KUKA KRL program: f1_Kuka_APT219T03S19.SRC

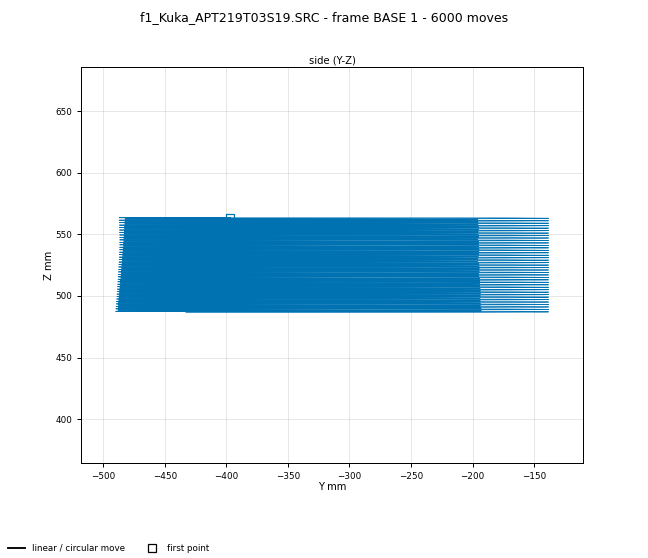
[picture p0: tool path of f1_Kuka_APT219T03S19.SRC in frame BASE 1, 6000 of 6001 moves have a stored position in this frame; points joined in program order, loops and branches not executed]
&ACCESS RVP
&REL 2
&PARAM TEMPLATE = C:\KRC\Roboter\Template\vorgabe
&PARAM EDITMASK = *
DEF f1_Kuka_APT219T03S19()


;FOLD INI;%{PE}%V3.2.0,%MKUKATPBASIS,%CINIT,%VCOMMON,%P
  ;FOLD BAS INI;%{E}%V3.2.0,%MKUKATPBASIS,%CINIT,%VINIT,%P
    GLOBAL INTERRUPT DECL 3 WHEN $STOPMESS==TRUE DO IR_STOPM ( )
    INTERRUPT ON 3
    BAS (#INITMOV,0 )
  ;ENDFOLD (BAS INI)
  ;FOLD USER INI;%{E}%V3.2.0,%MKUKATPUSER,%CINIT,%VINIT,%P
    ;Make your modifications here
  ;ENDFOLD (USER INI)
;ENDFOLD (INI)


;*** Make Null PTP Move
  PTP $pos_act

;*** Auto Load The Correct TOOL Data
  $tool=tool_data[3]

;*** Auto Load The Correct BASE Data
  $base=base_data[1]

  $ADVANCE = 5

;*** Restate Last Velocity
MMPM(30000.0)
SetRPM(6000)
LIN {X 0.052,Y -396.888,Z 563.591,A 0.000,B 0.000,C 90.000,E1 286.315} C_DIS
LIN {X 0.069,Y -413.808,Z 563.580,A 0.000,B 0.000,C 90.000,E1 284.356} C_DIS
LIN {X -0.094,Y -425.703,Z 563.572,A 0.000,B 0.000,C 90.000,E1 283.008} C_DIS
LIN {X 0.164,Y -434.823,Z 563.566,A 0.000,B 0.000,C 90.000,E1 281.895} C_DIS
LIN {X 0.106,Y -443.464,Z 563.560,A 0.000,B 0.000,C 90.000,E1 280.838} C_DIS
LIN {X -0.094,Y -449.609,Z 563.556,A 0.000,B 0.000,C 90.000,E1 280.074} C_DIS
LIN {X -0.070,Y -457.217,Z 563.550,A 0.000,B 0.000,C 90.000,E1 279.029} C_DIS
LIN {X -0.024,Y -464.281,Z 563.544,A 0.000,B 0.000,C 90.000,E1 277.992} C_DIS
LIN {X 0.173,Y -470.590,Z 563.539,A 0.000,B 0.000,C 90.000,E1 276.947} C_DIS
LIN {X -0.087,Y -476.108,Z 563.533,A 0.000,B 0.000,C 90.000,E1 275.967} C_DIS
LIN {X -0.149,Y -479.640,Z 563.529,A 0.000,B 0.000,C 90.000,E1 275.220} C_DIS
LIN {X 0.002,Y -481.624,Z 563.526,A 0.000,B 0.000,C 90.000,E1 274.702} C_DIS
LIN {X 0.124,Y -483.330,Z 563.523,A 0.000,B 0.000,C 90.000,E1 274.188} C_DIS
LIN {X -0.189,Y -484.732,Z 563.521,A 0.000,B 0.000,C 90.000,E1 273.726} C_DIS
LIN {X -0.041,Y -485.835,Z 563.518,A 0.000,B 0.000,C 90.000,E1 273.212} C_DIS
LIN {X 0.144,Y -486.619,Z 563.515,A 0.000,B 0.000,C 90.000,E1 272.694} C_DIS
LIN {X -0.175,Y -486.999,Z 563.512,A 0.000,B 0.000,C 90.000,E1 272.236} C_DIS
LIN {X 0.015,Y -486.990,Z 563.510,A 0.000,B 0.000,C 90.000,E1 271.718} C_DIS
LIN {X 0.189,Y -486.484,Z 563.507,A 0.000,B 0.000,C 90.000,E1 271.203} C_DIS
LIN {X -0.120,Y -485.459,Z 563.504,A 0.000,B 0.000,C 90.000,E1 270.745} C_DIS
LIN {X 0.053,Y -483.968,Z 563.501,A 0.000,B 0.000,C 90.000,E1 270.229} C_DIS
LIN {X 0.221,Y -481.805,Z 563.499,A 0.000,B 0.000,C 90.000,E1 269.714} C_DIS
LIN {X -0.102,Y -478.951,Z 563.496,A 0.000,B 0.000,C 90.000,E1 269.255} C_DIS
LIN {X 0.035,Y -475.279,Z 563.493,A 0.000,B 0.000,C 90.000,E1 268.740} C_DIS
LIN {X 0.149,Y -470.579,Z 563.490,A 0.000,B 0.000,C 90.000,E1 268.224} C_DIS
LIN {X -0.010,Y -467.817,Z 563.489,A 0.000,B 0.000,C 90.000,E1 267.993} C_DIS
LIN {X -0.053,Y -461.679,Z 563.486,A 0.000,B 0.000,C 90.000,E1 267.535} C_DIS
LIN {X 0.032,Y -454.984,Z 563.484,A 0.000,B 0.000,C 90.000,E1 267.135} C_DIS
LIN {X -0.209,Y -447.920,Z 563.482,A 0.000,B 0.000,C 90.000,E1 266.846} C_DIS
LIN {X 0.025,Y -440.647,Z 563.481,A 0.000,B 0.000,C 90.000,E1 266.560} C_DIS
LIN {X 0.215,Y -432.943,Z 563.480,A 0.000,B 0.000,C 90.000,E1 266.331} C_DIS
LIN {X -0.106,Y -424.380,Z 563.479,A 0.000,B 0.000,C 90.000,E1 266.216} C_DIS
LIN {X -0.080,Y -413.364,Z 563.478,A 0.000,B 0.000,C 90.000,E1 266.102} C_DIS
LIN {X 0.171,Y -408.029,Z 563.478,A 0.000,B 0.000,C 90.000,E1 266.045} C_DIS
LIN {X 0.041,Y -180.922,Z 563.478,A 0.000,B 0.000,C 90.000,E1 266.045} C_DIS
LIN {X 0.082,Y -180.869,Z 563.472,A 0.000,B 0.000,C 90.000,E1 265.008} C_DIS
LIN {X -0.015,Y -178.930,Z 563.443,A 0.000,B 0.000,C 90.000,E1 259.803} C_DIS
LIN {X 0.023,Y -175.977,Z 563.415,A 0.000,B 0.000,C 90.000,E1 254.700} C_DIS
LIN {X -0.032,Y -175.468,Z 563.410,A 0.000,B 0.000,C 90.000,E1 253.866} C_DIS
LIN {X 0.025,Y -172.217,Z 563.387,A 0.000,B 0.000,C 90.000,E1 249.571} C_DIS
LIN {X 0.002,Y -171.693,Z 563.382,A 0.000,B 0.000,C 90.000,E1 248.720} C_DIS
LIN {X 0.078,Y -167.287,Z 563.353,A 0.000,B 0.000,C 90.000,E1 243.512} C_DIS
LIN {X 0.011,Y -166.663,Z 563.348,A 0.000,B 0.000,C 90.000,E1 242.666} C_DIS
LIN {X -0.073,Y -162.646,Z 563.324,A 0.000,B 0.000,C 90.000,E1 238.329} C_DIS
LIN {X -0.011,Y -161.335,Z 563.314,A 0.000,B 0.000,C 90.000,E1 236.548} C_DIS
LIN {X 0.033,Y -157.330,Z 563.290,A 0.000,B 0.000,C 90.000,E1 232.110} C_DIS
LIN {X -0.034,Y -155.312,Z 563.275,A 0.000,B 0.000,C 90.000,E1 229.461} C_DIS
LIN {X 0.003,Y -151.668,Z 563.250,A 0.000,B 0.000,C 90.000,E1 224.960} C_DIS
LIN {X 0.047,Y -150.534,Z 563.240,A 0.000,B 0.000,C 90.000,E1 223.137} C_DIS
LIN {X -0.022,Y -147.259,Z 563.215,A 0.000,B 0.000,C 90.000,E1 218.624} C_DIS
LIN {X 0.034,Y -145.285,Z 563.194,A 0.000,B 0.000,C 90.000,E1 214.945} C_DIS
LIN {X 0.068,Y -142.386,Z 563.164,A 0.000,B 0.000,C 90.000,E1 209.411} C_DIS
LIN {X -0.010,Y -141.364,Z 563.148,A 0.000,B 0.000,C 90.000,E1 206.668} C_DIS
LIN {X -0.032,Y -139.344,Z 563.112,A 0.000,B 0.000,C 90.000,E1 200.174} C_DIS
LIN {X -0.026,Y -139.013,Z 563.102,A 0.000,B 0.000,C 90.000,E1 198.308} C_DIS
LIN {X -0.031,Y -138.342,Z 563.055,A 0.000,B 0.000,C 90.000,E1 189.905} C_DIS
LIN {X -0.011,Y -139.397,Z 563.008,A 0.000,B 0.000,C 90.000,E1 181.489} C_DIS
LIN {X 0.043,Y -141.299,Z 562.972,A 0.000,B 0.000,C 90.000,E1 174.951} C_DIS
LIN {X 0.000,Y -142.661,Z 562.957,A 0.000,B 0.000,C 90.000,E1 172.186} C_DIS
LIN {X -0.050,Y -145.005,Z 562.931,A 0.000,B 0.000,C 90.000,E1 167.589} C_DIS
LIN {X -0.061,Y -147.631,Z 562.911,A 0.000,B 0.000,C 90.000,E1 163.921} C_DIS
LIN {X 0.017,Y -150.261,Z 562.890,A 0.000,B 0.000,C 90.000,E1 160.242} C_DIS
LIN {X 0.031,Y -153.661,Z 562.870,A 0.000,B 0.000,C 90.000,E1 156.613} C_DIS
LIN {X 0.088,Y -157.075,Z 562.850,A 0.000,B 0.000,C 90.000,E1 152.999} C_DIS
LIN {X 0.026,Y -161.209,Z 562.830,A 0.000,B 0.000,C 90.000,E1 149.459} C_DIS
LIN {X -0.025,Y -163.299,Z 562.821,A 0.000,B 0.000,C 90.000,E1 147.709} C_DIS
LIN {X -0.016,Y -167.747,Z 562.801,A 0.000,B 0.000,C 90.000,E1 144.196} C_DIS
LIN {X -0.104,Y -171.564,Z 562.787,A 0.000,B 0.000,C 90.000,E1 141.618} C_DIS
LIN {X -0.063,Y -176.509,Z 562.767,A 0.000,B 0.000,C 90.000,E1 138.162} C_DIS
LIN {X 0.062,Y -180.807,Z 562.753,A 0.000,B 0.000,C 90.000,E1 135.567} C_DIS
LIN {X 0.048,Y -186.216,Z 562.735,A 0.000,B 0.000,C 90.000,E1 132.204} C_DIS
LIN {X 0.001,Y -191.316,Z 562.719,A 0.000,B 0.000,C 90.000,E1 129.439} C_DIS
LIN {X 0.030,Y -191.697,Z 562.718,A 0.000,B 0.000,C 90.000,E1 129.197} C_DIS
LIN {X -0.009,Y -289.306,Z 562.718,A 0.000,B 0.000,C 90.000,E1 129.197} C_DIS
LIN {X -0.167,Y -290.832,Z 562.718,A 0.000,B 0.000,C 90.000,E1 129.197} C_DIS
LIN {X -0.087,Y -295.851,Z 562.716,A 0.000,B 0.000,C 90.000,E1 128.910} C_DIS
LIN {X 0.094,Y -299.087,Z 562.714,A 0.000,B 0.000,C 90.000,E1 128.543} C_DIS
LIN {X 0.060,Y -302.684,Z 562.711,A 0.000,B 0.000,C 90.000,E1 127.971} C_DIS
LIN {X 0.009,Y -304.123,Z 562.709,A 0.000,B 0.000,C 90.000,E1 127.649} C_DIS
LIN {X 0.011,Y -305.255,Z 562.707,A 0.000,B 0.000,C 90.000,E1 127.317} C_DIS
LIN {X 0.076,Y -314.947,Z 562.689,A 0.000,B 0.000,C 90.000,E1 124.040} C_DIS
LIN {X -0.069,Y -324.944,Z 562.673,A 0.000,B 0.000,C 90.000,E1 121.180} C_DIS
LIN {X -0.154,Y -336.268,Z 562.657,A 0.000,B 0.000,C 90.000,E1 118.359} C_DIS
LIN {X 0.090,Y -349.018,Z 562.642,A 0.000,B 0.000,C 90.000,E1 115.540} C_DIS
LIN {X 0.027,Y -361.644,Z 562.629,A 0.000,B 0.000,C 90.000,E1 113.131} C_DIS
LIN {X -0.160,Y -375.580,Z 562.615,A 0.000,B 0.000,C 90.000,E1 110.791} C_DIS
LIN {X 0.233,Y -390.927,Z 562.602,A 0.000,B 0.000,C 90.000,E1 108.417} C_DIS
LIN {X -0.096,Y -407.797,Z 562.590,A 0.000,B 0.000,C 90.000,E1 106.205} C_DIS
LIN {X -0.131,Y -426.314,Z 562.578,A 0.000,B 0.000,C 90.000,E1 104.008} C_DIS
LIN {X 0.058,Y -446.220,Z 562.566,A 0.000,B 0.000,C 90.000,E1 101.883} C_DIS
LIN {X 0.002,Y -466.729,Z 562.555,A 0.000,B 0.000,C 90.000,E1 99.962} C_DIS
LIN {X 0.122,Y -474.560,Z 562.552,A 0.000,B 0.000,C 90.000,E1 99.265} C_DIS
LIN {X 0.213,Y -476.741,Z 562.550,A 0.000,B 0.000,C 90.000,E1 99.029} C_DIS
LIN {X -0.243,Y -478.398,Z 562.549,A 0.000,B 0.000,C 90.000,E1 98.859} C_DIS
LIN {X 0.100,Y -479.812,Z 562.548,A 0.000,B 0.000,C 90.000,E1 98.568} C_DIS
LIN {X -0.103,Y -480.863,Z 562.546,A 0.000,B 0.000,C 90.000,E1 98.341} C_DIS
LIN {X 0.126,Y -482.084,Z 562.544,A 0.000,B 0.000,C 90.000,E1 97.814} C_DIS
LIN {X -0.187,Y -482.293,Z 562.541,A 0.000,B 0.000,C 90.000,E1 97.352} C_DIS
LIN {X -0.012,Y -481.523,Z 562.538,A 0.000,B 0.000,C 90.000,E1 96.834} C_DIS
LIN {X 0.162,Y -479.651,Z 562.535,A 0.000,B 0.000,C 90.000,E1 96.315} C_DIS
LIN {X -0.016,Y -478.187,Z 562.534,A 0.000,B 0.000,C 90.000,E1 96.087} C_DIS
LIN {X 0.053,Y -459.322,Z 562.520,A 0.000,B 0.000,C 90.000,E1 93.555} C_DIS
LIN {X -0.137,Y -450.857,Z 562.513,A 0.000,B 0.000,C 90.000,E1 92.293} C_DIS
LIN {X 0.013,Y -435.844,Z 562.498,A 0.000,B 0.000,C 90.000,E1 89.656} C_DIS
LIN {X -0.085,Y -428.020,Z 562.491,A 0.000,B 0.000,C 90.000,E1 88.339} C_DIS
LIN {X 0.183,Y -413.667,Z 562.477,A 0.000,B 0.000,C 90.000,E1 85.869} C_DIS
LIN {X 0.104,Y -399.695,Z 562.463,A 0.000,B 0.000,C 90.000,E1 83.394} C_DIS
LIN {X 0.099,Y -387.583,Z 562.451,A 0.000,B 0.000,C 90.000,E1 81.141} C_DIS
LIN {X -0.089,Y -377.024,Z 562.440,A 0.000,B 0.000,C 90.000,E1 79.162} C_DIS
LIN {X -0.060,Y -366.493,Z 562.428,A 0.000,B 0.000,C 90.000,E1 77.117} C_DIS
LIN {X -0.085,Y -356.606,Z 562.417,A 0.000,B 0.000,C 90.000,E1 75.046} C_DIS
LIN {X 0.053,Y -345.316,Z 562.402,A 0.000,B 0.000,C 90.000,E1 72.308} C_DIS
LIN {X -0.122,Y -335.188,Z 562.386,A 0.000,B 0.000,C 90.000,E1 69.571} C_DIS
LIN {X 0.025,Y -323.108,Z 562.366,A 0.000,B 0.000,C 90.000,E1 65.793} C_DIS
LIN {X -0.017,Y -315.556,Z 562.351,A 0.000,B 0.000,C 90.000,E1 63.256} C_DIS
LIN {X 0.034,Y -308.153,Z 562.337,A 0.000,B 0.000,C 90.000,E1 60.667} C_DIS
LIN {X -0.066,Y -300.848,Z 562.323,A 0.000,B 0.000,C 90.000,E1 58.074} C_DIS
LIN {X -0.113,Y -292.016,Z 562.304,A 0.000,B 0.000,C 90.000,E1 54.769} C_DIS
LIN {X -0.040,Y -285.310,Z 562.289,A 0.000,B 0.000,C 90.000,E1 52.065} C_DIS
LIN {X 0.138,Y -280.088,Z 562.278,A 0.000,B 0.000,C 90.000,E1 49.989} C_DIS
LIN {X -0.001,Y -276.380,Z 562.270,A 0.000,B 0.000,C 90.000,E1 48.647} C_DIS
LIN {X -0.005,Y -272.388,Z 562.263,A 0.000,B 0.000,C 90.000,E1 47.268} C_DIS
LIN {X 0.003,Y -266.989,Z 562.253,A 0.000,B 0.000,C 90.000,E1 45.526} C_DIS
LIN {X -0.032,Y -259.975,Z 562.241,A 0.000,B 0.000,C 90.000,E1 43.419} C_DIS
LIN {X 0.052,Y -249.600,Z 562.223,A 0.000,B 0.000,C 90.000,E1 40.172} C_DIS
LIN {X 0.110,Y -240.982,Z 562.207,A 0.000,B 0.000,C 90.000,E1 37.237} C_DIS
LIN {X 0.066,Y -233.091,Z 562.191,A 0.000,B 0.000,C 90.000,E1 34.278} C_DIS
LIN {X 0.077,Y -225.826,Z 562.174,A 0.000,B 0.000,C 90.000,E1 31.258} C_DIS
LIN {X -0.054,Y -219.357,Z 562.157,A 0.000,B 0.000,C 90.000,E1 28.231} C_DIS
LIN {X 0.039,Y -213.668,Z 562.140,A 0.000,B 0.000,C 90.000,E1 25.103} C_DIS
LIN {X 0.009,Y -208.726,Z 562.122,A 0.000,B 0.000,C 90.000,E1 21.972} C_DIS
LIN {X 0.015,Y -203.999,Z 562.100,A 0.000,B 0.000,C 90.000,E1 18.000} C_DIS
LIN {X -0.046,Y -200.157,Z 562.078,A 0.000,B 0.000,C 90.000,E1 14.008} C_DIS
LIN {X -0.030,Y -197.066,Z 562.051,A 0.000,B 0.000,C 90.000,E1 9.151} C_DIS
LIN {X 0.022,Y -195.867,Z 561.984,A 0.000,B 0.000,C 90.000,E1 357.078} C_DIS
LIN {X 0.040,Y -198.513,Z 561.952,A 0.000,B 0.000,C 90.000,E1 351.376} C_DIS
LIN {X 0.008,Y -202.175,Z 561.925,A 0.000,B 0.000,C 90.000,E1 346.533} C_DIS
LIN {X 0.058,Y -207.047,Z 561.898,A 0.000,B 0.000,C 90.000,E1 341.710} C_DIS
LIN {X 0.063,Y -211.977,Z 561.876,A 0.000,B 0.000,C 90.000,E1 337.741} C_DIS
LIN {X -0.041,Y -217.541,Z 561.855,A 0.000,B 0.000,C 90.000,E1 333.845} C_DIS
LIN {X 0.027,Y -223.698,Z 561.833,A 0.000,B 0.000,C 90.000,E1 329.950} C_DIS
LIN {X -0.021,Y -230.451,Z 561.812,A 0.000,B 0.000,C 90.000,E1 326.135} C_DIS
LIN {X 0.026,Y -237.729,Z 561.791,A 0.000,B 0.000,C 90.000,E1 322.351} C_DIS
LIN {X -0.026,Y -245.514,Z 561.770,A 0.000,B 0.000,C 90.000,E1 318.647} C_DIS
LIN {X -0.071,Y -254.238,Z 561.750,A 0.000,B 0.000,C 90.000,E1 315.000} C_DIS
LIN {X 0.016,Y -264.417,Z 561.730,A 0.000,B 0.000,C 90.000,E1 311.391} C_DIS
LIN {X 0.037,Y -274.703,Z 561.712,A 0.000,B 0.000,C 90.000,E1 308.222} C_DIS
LIN {X -0.158,Y -287.628,Z 561.693,A 0.000,B 0.000,C 90.000,E1 304.818} C_DIS
LIN {X 0.067,Y -301.962,Z 561.675,A 0.000,B 0.000,C 90.000,E1 301.416} C_DIS
LIN {X 0.029,Y -317.471,Z 561.656,A 0.000,B 0.000,C 90.000,E1 298.153} C_DIS
LIN {X 0.090,Y -330.845,Z 561.642,A 0.000,B 0.000,C 90.000,E1 295.591} C_DIS
LIN {X 0.085,Y -341.774,Z 561.632,A 0.000,B 0.000,C 90.000,E1 293.718} C_DIS
LIN {X 0.001,Y -355.893,Z 561.620,A 0.000,B 0.000,C 90.000,E1 291.589} C_DIS
LIN {X 0.112,Y -378.082,Z 561.603,A 0.000,B 0.000,C 90.000,E1 288.598} C_DIS
LIN {X -0.024,Y -396.955,Z 561.591,A 0.000,B 0.000,C 90.000,E1 286.315} C_DIS
LIN {X -0.027,Y -413.945,Z 561.580,A 0.000,B 0.000,C 90.000,E1 284.356} C_DIS
LIN {X -0.191,Y -425.861,Z 561.572,A 0.000,B 0.000,C 90.000,E1 283.008} C_DIS
LIN {X -0.168,Y -437.191,Z 561.565,A 0.000,B 0.000,C 90.000,E1 281.658} C_DIS
LIN {X -0.206,Y -445.725,Z 561.559,A 0.000,B 0.000,C 90.000,E1 280.602} C_DIS
LIN {X -0.229,Y -453.687,Z 561.553,A 0.000,B 0.000,C 90.000,E1 279.557} C_DIS
LIN {X -0.155,Y -461.011,Z 561.547,A 0.000,B 0.000,C 90.000,E1 278.511} C_DIS
LIN {X 0.001,Y -467.696,Z 561.542,A 0.000,B 0.000,C 90.000,E1 277.466} C_DIS
LIN {X 0.176,Y -473.606,Z 561.536,A 0.000,B 0.000,C 90.000,E1 276.429} C_DIS
LIN {X 0.094,Y -477.501,Z 561.532,A 0.000,B 0.000,C 90.000,E1 275.682} C_DIS
LIN {X 0.235,Y -479.763,Z 561.529,A 0.000,B 0.000,C 90.000,E1 275.163} C_DIS
LIN {X -0.091,Y -481.699,Z 561.526,A 0.000,B 0.000,C 90.000,E1 274.702} C_DIS
LIN {X 0.031,Y -483.375,Z 561.523,A 0.000,B 0.000,C 90.000,E1 274.188} C_DIS
LIN {X 0.201,Y -484.766,Z 561.521,A 0.000,B 0.000,C 90.000,E1 273.669} C_DIS
LIN {X -0.134,Y -485.861,Z 561.518,A 0.000,B 0.000,C 90.000,E1 273.212} C_DIS
LIN {X 0.051,Y -486.604,Z 561.515,A 0.000,B 0.000,C 90.000,E1 272.694} C_DIS
LIN {X 0.219,Y -486.963,Z 561.512,A 0.000,B 0.000,C 90.000,E1 272.178} C_DIS
LIN {X -0.079,Y -486.910,Z 561.510,A 0.000,B 0.000,C 90.000,E1 271.718} C_DIS
LIN {X 0.096,Y -486.380,Z 561.507,A 0.000,B 0.000,C 90.000,E1 271.203} C_DIS
LIN {X -0.213,Y -485.369,Z 561.504,A 0.000,B 0.000,C 90.000,E1 270.745} C_DIS
LIN {X -0.040,Y -483.839,Z 561.501,A 0.000,B 0.000,C 90.000,E1 270.229} C_DIS
LIN {X 0.127,Y -481.713,Z 561.498,A 0.000,B 0.000,C 90.000,E1 269.714} C_DIS
LIN {X -0.195,Y -478.851,Z 561.496,A 0.000,B 0.000,C 90.000,E1 269.255} C_DIS
LIN {X 0.111,Y -477.136,Z 561.494,A 0.000,B 0.000,C 90.000,E1 268.969} C_DIS
LIN {X -0.238,Y -472.936,Z 561.492,A 0.000,B 0.000,C 90.000,E1 268.511} C_DIS
LIN {X 0.055,Y -470.464,Z 561.490,A 0.000,B 0.000,C 90.000,E1 268.224} C_DIS
LIN {X 0.210,Y -464.565,Z 561.487,A 0.000,B 0.000,C 90.000,E1 267.707} C_DIS
LIN {X -0.051,Y -457.943,Z 561.485,A 0.000,B 0.000,C 90.000,E1 267.306} C_DIS
LIN {X -0.150,Y -450.861,Z 561.483,A 0.000,B 0.000,C 90.000,E1 266.963} C_DIS
LIN {X -0.103,Y -443.585,Z 561.481,A 0.000,B 0.000,C 90.000,E1 266.674} C_DIS
LIN {X -0.079,Y -436.161,Z 561.480,A 0.000,B 0.000,C 90.000,E1 266.445} C_DIS
LIN {X -0.122,Y -428.114,Z 561.479,A 0.000,B 0.000,C 90.000,E1 266.274} C_DIS
LIN {X 0.185,Y -418.501,Z 561.479,A 0.000,B 0.000,C 90.000,E1 266.102} C_DIS
LIN {X -0.209,Y -409.834,Z 561.478,A 0.000,B 0.000,C 90.000,E1 266.102} C_DIS
LIN {X 0.121,Y -403.931,Z 561.478,A 0.000,B 0.000,C 90.000,E1 266.045} C_DIS
LIN {X 0.020,Y -180.922,Z 561.478,A 0.000,B 0.000,C 90.000,E1 266.045} C_DIS
LIN {X 0.061,Y -180.868,Z 561.472,A 0.000,B 0.000,C 90.000,E1 265.008} C_DIS
LIN {X -0.036,Y -178.928,Z 561.443,A 0.000,B 0.000,C 90.000,E1 259.803} C_DIS
LIN {X 0.003,Y -175.974,Z 561.415,A 0.000,B 0.000,C 90.000,E1 254.700} C_DIS
LIN {X -0.052,Y -175.462,Z 561.410,A 0.000,B 0.000,C 90.000,E1 253.866} C_DIS
LIN {X 0.005,Y -172.213,Z 561.387,A 0.000,B 0.000,C 90.000,E1 249.571} C_DIS
LIN {X -0.017,Y -171.689,Z 561.382,A 0.000,B 0.000,C 90.000,E1 248.720} C_DIS
LIN {X -0.026,Y -167.915,Z 561.358,A 0.000,B 0.000,C 90.000,E1 244.409} C_DIS
LIN {X -0.009,Y -166.657,Z 561.348,A 0.000,B 0.000,C 90.000,E1 242.666} C_DIS
LIN {X 0.046,Y -162.641,Z 561.324,A 0.000,B 0.000,C 90.000,E1 238.280} C_DIS
LIN {X -0.030,Y -161.329,Z 561.314,A 0.000,B 0.000,C 90.000,E1 236.548} C_DIS
LIN {X 0.013,Y -157.324,Z 561.290,A 0.000,B 0.000,C 90.000,E1 232.110} C_DIS
LIN {X -0.054,Y -155.305,Z 561.275,A 0.000,B 0.000,C 90.000,E1 229.461} C_DIS
LIN {X -0.015,Y -151.664,Z 561.250,A 0.000,B 0.000,C 90.000,E1 224.960} C_DIS
LIN {X 0.030,Y -150.530,Z 561.240,A 0.000,B 0.000,C 90.000,E1 223.137} C_DIS
LIN {X -0.040,Y -147.255,Z 561.214,A 0.000,B 0.000,C 90.000,E1 218.624} C_DIS
LIN {X 0.017,Y -145.280,Z 561.194,A 0.000,B 0.000,C 90.000,E1 214.945} C_DIS
LIN {X 0.049,Y -142.383,Z 561.164,A 0.000,B 0.000,C 90.000,E1 209.411} C_DIS
LIN {X -0.027,Y -141.361,Z 561.148,A 0.000,B 0.000,C 90.000,E1 206.668} C_DIS
LIN {X -0.049,Y -139.343,Z 561.112,A 0.000,B 0.000,C 90.000,E1 200.174} C_DIS
LIN {X -0.043,Y -139.012,Z 561.102,A 0.000,B 0.000,C 90.000,E1 198.308} C_DIS
LIN {X -0.049,Y -138.341,Z 561.055,A 0.000,B 0.000,C 90.000,E1 189.905} C_DIS
LIN {X -0.028,Y -139.398,Z 561.008,A 0.000,B 0.000,C 90.000,E1 181.489} C_DIS
LIN {X 0.025,Y -141.302,Z 560.972,A 0.000,B 0.000,C 90.000,E1 174.951} C_DIS
LIN {X -0.018,Y -142.663,Z 560.957,A 0.000,B 0.000,C 90.000,E1 172.186} C_DIS
LIN {X -0.068,Y -145.009,Z 560.931,A 0.000,B 0.000,C 90.000,E1 167.589} C_DIS
LIN {X -0.079,Y -147.636,Z 560.911,A 0.000,B 0.000,C 90.000,E1 163.921} C_DIS
LIN {X -0.002,Y -150.267,Z 560.890,A 0.000,B 0.000,C 90.000,E1 160.242} C_DIS
LIN {X 0.012,Y -153.668,Z 560.870,A 0.000,B 0.000,C 90.000,E1 156.613} C_DIS
LIN {X 0.068,Y -157.082,Z 560.850,A 0.000,B 0.000,C 90.000,E1 152.999} C_DIS
LIN {X 0.006,Y -161.217,Z 560.830,A 0.000,B 0.000,C 90.000,E1 149.459} C_DIS
LIN {X -0.045,Y -163.307,Z 560.820,A 0.000,B 0.000,C 90.000,E1 147.709} C_DIS
LIN {X -0.036,Y -167.756,Z 560.801,A 0.000,B 0.000,C 90.000,E1 144.196} C_DIS
LIN {X -0.018,Y -171.572,Z 560.787,A 0.000,B 0.000,C 90.000,E1 141.582} C_DIS
LIN {X -0.083,Y -176.520,Z 560.767,A 0.000,B 0.000,C 90.000,E1 138.162} C_DIS
LIN {X 0.041,Y -180.818,Z 560.753,A 0.000,B 0.000,C 90.000,E1 135.567} C_DIS
LIN {X 0.027,Y -186.228,Z 560.734,A 0.000,B 0.000,C 90.000,E1 132.204} C_DIS
LIN {X -0.020,Y -191.327,Z 560.719,A 0.000,B 0.000,C 90.000,E1 129.439} C_DIS
LIN {X -0.028,Y -191.726,Z 560.718,A 0.000,B 0.000,C 90.000,E1 129.197} C_DIS
LIN {X -0.096,Y -289.223,Z 560.718,A 0.000,B 0.000,C 90.000,E1 129.197} C_DIS
LIN {X 0.024,Y -290.403,Z 560.718,A 0.000,B 0.000,C 90.000,E1 129.152} C_DIS
LIN {X -0.120,Y -295.730,Z 560.716,A 0.000,B 0.000,C 90.000,E1 128.910} C_DIS
LIN {X -0.077,Y -298.871,Z 560.714,A 0.000,B 0.000,C 90.000,E1 128.588} C_DIS
LIN {X -0.050,Y -302.502,Z 560.711,A 0.000,B 0.000,C 90.000,E1 128.016} C_DIS
LIN {X -0.049,Y -303.987,Z 560.709,A 0.000,B 0.000,C 90.000,E1 127.684} C_DIS
LIN {X -0.104,Y -305.155,Z 560.707,A 0.000,B 0.000,C 90.000,E1 127.363} C_DIS
LIN {X -0.174,Y -315.897,Z 560.688,A 0.000,B 0.000,C 90.000,E1 123.785} C_DIS
LIN {X -0.015,Y -326.028,Z 560.672,A 0.000,B 0.000,C 90.000,E1 120.875} C_DIS
LIN {X 0.109,Y -337.493,Z 560.656,A 0.000,B 0.000,C 90.000,E1 118.025} C_DIS
LIN {X -0.078,Y -350.399,Z 560.640,A 0.000,B 0.000,C 90.000,E1 115.283} C_DIS
LIN {X 0.078,Y -363.172,Z 560.627,A 0.000,B 0.000,C 90.000,E1 112.845} C_DIS
LIN {X 0.078,Y -377.267,Z 560.614,A 0.000,B 0.000,C 90.000,E1 110.482} C_DIS
LIN {X 0.026,Y -392.784,Z 560.601,A 0.000,B 0.000,C 90.000,E1 108.181} C_DIS
LIN {X -0.150,Y -409.839,Z 560.589,A 0.000,B 0.000,C 90.000,E1 105.953} C_DIS
LIN {X 0.163,Y -428.557,Z 560.576,A 0.000,B 0.000,C 90.000,E1 103.716} C_DIS
LIN {X -0.021,Y -448.564,Z 560.565,A 0.000,B 0.000,C 90.000,E1 101.658} C_DIS
LIN {X 0.169,Y -469.133,Z 560.554,A 0.000,B 0.000,C 90.000,E1 99.726} C_DIS
LIN {X -0.220,Y -474.356,Z 560.552,A 0.000,B 0.000,C 90.000,E1 99.321} C_DIS
LIN {X -0.180,Y -476.594,Z 560.550,A 0.000,B 0.000,C 90.000,E1 99.095} C_DIS
LIN {X -0.064,Y -478.292,Z 560.549,A 0.000,B 0.000,C 90.000,E1 98.859} C_DIS
LIN {X -0.195,Y -479.761,Z 560.548,A 0.000,B 0.000,C 90.000,E1 98.624} C_DIS
LIN {X 0.078,Y -480.858,Z 560.546,A 0.000,B 0.000,C 90.000,E1 98.341} C_DIS
LIN {X -0.172,Y -482.152,Z 560.544,A 0.000,B 0.000,C 90.000,E1 97.871} C_DIS
LIN {X -0.007,Y -482.427,Z 560.541,A 0.000,B 0.000,C 90.000,E1 97.352} C_DIS
LIN {X 0.168,Y -481.727,Z 560.538,A 0.000,B 0.000,C 90.000,E1 96.834} C_DIS
LIN {X -0.135,Y -479.939,Z 560.535,A 0.000,B 0.000,C 90.000,E1 96.372} C_DIS
LIN {X 0.164,Y -478.531,Z 560.534,A 0.000,B 0.000,C 90.000,E1 96.087} C_DIS
LIN {X -0.195,Y -468.939,Z 560.527,A 0.000,B 0.000,C 90.000,E1 94.878} C_DIS
LIN {X -0.176,Y -456.144,Z 560.517,A 0.000,B 0.000,C 90.000,E1 93.094} C_DIS
LIN {X -0.210,Y -446.470,Z 560.508,A 0.000,B 0.000,C 90.000,E1 91.547} C_DIS
LIN {X 0.199,Y -436.077,Z 560.498,A 0.000,B 0.000,C 90.000,E1 89.656} C_DIS
LIN {X 0.101,Y -428.255,Z 560.491,A 0.000,B 0.000,C 90.000,E1 88.339} C_DIS
LIN {X -0.045,Y -413.902,Z 560.477,A 0.000,B 0.000,C 90.000,E1 85.927} C_DIS
LIN {X -0.108,Y -399.903,Z 560.464,A 0.000,B 0.000,C 90.000,E1 83.451} C_DIS
LIN {X -0.100,Y -387.767,Z 560.451,A 0.000,B 0.000,C 90.000,E1 81.197} C_DIS
LIN {X 0.094,Y -377.178,Z 560.440,A 0.000,B 0.000,C 90.000,E1 79.162} C_DIS
LIN {X 0.120,Y -366.618,Z 560.429,A 0.000,B 0.000,C 90.000,E1 77.117} C_DIS
LIN {X 0.043,Y -358.055,Z 560.419,A 0.000,B 0.000,C 90.000,E1 75.353} C_DIS
LIN {X -0.120,Y -346.603,Z 560.404,A 0.000,B 0.000,C 90.000,E1 72.670} C_DIS
LIN {X 0.064,Y -337.419,Z 560.390,A 0.000,B 0.000,C 90.000,E1 70.188} C_DIS
LIN {X -0.086,Y -327.084,Z 560.373,A 0.000,B 0.000,C 90.000,E1 67.102} C_DIS
LIN {X 0.128,Y -319.418,Z 560.359,A 0.000,B 0.000,C 90.000,E1 64.537} C_DIS
LIN {X 0.128,Y -311.945,Z 560.344,A 0.000,B 0.000,C 90.000,E1 61.975} C_DIS
LIN {X -0.036,Y -304.594,Z 560.330,A 0.000,B 0.000,C 90.000,E1 59.410} C_DIS
LIN {X -0.068,Y -297.336,Z 560.315,A 0.000,B 0.000,C 90.000,E1 56.786} C_DIS
LIN {X 0.107,Y -288.746,Z 560.297,A 0.000,B 0.000,C 90.000,E1 53.417} C_DIS
LIN {X -0.001,Y -283.649,Z 560.286,A 0.000,B 0.000,C 90.000,E1 51.412} C_DIS
LIN {X -0.068,Y -278.319,Z 560.274,A 0.000,B 0.000,C 90.000,E1 49.380} C_DIS
LIN {X -0.043,Y -274.473,Z 560.267,A 0.000,B 0.000,C 90.000,E1 48.000} C_DIS
LIN {X -0.066,Y -270.342,Z 560.259,A 0.000,B 0.000,C 90.000,E1 46.620} C_DIS
LIN {X 0.097,Y -264.739,Z 560.249,A 0.000,B 0.000,C 90.000,E1 44.838} C_DIS
LIN {X 0.084,Y -255.313,Z 560.233,A 0.000,B 0.000,C 90.000,E1 42.000} C_DIS
LIN {X 0.054,Y -245.230,Z 560.215,A 0.000,B 0.000,C 90.000,E1 38.749} C_DIS
LIN {X 0.059,Y -236.960,Z 560.199,A 0.000,B 0.000,C 90.000,E1 35.804} C_DIS
LIN {X -0.024,Y -229.356,Z 560.182,A 0.000,B 0.000,C 90.000,E1 32.832} C_DIS
LIN {X -0.032,Y -222.480,Z 560.165,A 0.000,B 0.000,C 90.000,E1 29.795} C_DIS
LIN {X 0.040,Y -216.408,Z 560.148,A 0.000,B 0.000,C 90.000,E1 26.693} C_DIS
LIN {X -0.030,Y -211.090,Z 560.131,A 0.000,B 0.000,C 90.000,E1 23.590} C_DIS
LIN {X -0.013,Y -206.702,Z 560.113,A 0.000,B 0.000,C 90.000,E1 20.429} C_DIS
LIN {X -0.010,Y -202.311,Z 560.091,A 0.000,B 0.000,C 90.000,E1 16.441} C_DIS
LIN {X 0.015,Y -198.944,Z 560.069,A 0.000,B 0.000,C 90.000,E1 12.411} C_DIS
LIN {X 0.061,Y -196.083,Z 560.037,A 0.000,B 0.000,C 90.000,E1 6.720} C_DIS
LIN {X 0.070,Y -195.621,Z 559.988,A 0.000,B 0.000,C 90.000,E1 357.879} C_DIS
LIN {X 0.045,Y -197.986,Z 559.957,A 0.000,B 0.000,C 90.000,E1 352.186} C_DIS
LIN {X -0.042,Y -201.455,Z 559.930,A 0.000,B 0.000,C 90.000,E1 347.353} C_DIS
LIN {X -0.072,Y -206.144,Z 559.903,A 0.000,B 0.000,C 90.000,E1 342.543} C_DIS
LIN {X 0.032,Y -210.905,Z 559.881,A 0.000,B 0.000,C 90.000,E1 338.539} C_DIS
LIN {X 0.096,Y -216.339,Z 559.859,A 0.000,B 0.000,C 90.000,E1 334.588} C_DIS
LIN {X 0.036,Y -222.383,Z 559.837,A 0.000,B 0.000,C 90.000,E1 330.717} C_DIS
LIN {X -0.098,Y -229.018,Z 559.816,A 0.000,B 0.000,C 90.000,E1 326.914} C_DIS
LIN {X -0.102,Y -236.230,Z 559.795,A 0.000,B 0.000,C 90.000,E1 323.130} C_DIS
LIN {X -0.010,Y -243.881,Z 559.774,A 0.000,B 0.000,C 90.000,E1 319.380} C_DIS
LIN {X -0.093,Y -252.380,Z 559.754,A 0.000,B 0.000,C 90.000,E1 315.729} C_DIS
LIN {X 0.068,Y -261.223,Z 559.736,A 0.000,B 0.000,C 90.000,E1 312.447} C_DIS
LIN {X 0.077,Y -272.289,Z 559.716,A 0.000,B 0.000,C 90.000,E1 308.910} C_DIS
LIN {X -0.016,Y -284.919,Z 559.697,A 0.000,B 0.000,C 90.000,E1 305.471} C_DIS
LIN {X 0.042,Y -298.966,Z 559.678,A 0.000,B 0.000,C 90.000,E1 302.084} C_DIS
LIN {X -0.092,Y -314.190,Z 559.660,A 0.000,B 0.000,C 90.000,E1 298.821} C_DIS
LIN {X -0.021,Y -329.010,Z 559.644,A 0.000,B 0.000,C 90.000,E1 295.924} C_DIS
LIN {X 0.078,Y -339.785,Z 559.634,A 0.000,B 0.000,C 90.000,E1 294.027} C_DIS
LIN {X -0.044,Y -353.728,Z 559.622,A 0.000,B 0.000,C 90.000,E1 291.897} C_DIS
LIN {X -0.103,Y -373.479,Z 559.607,A 0.000,B 0.000,C 90.000,E1 289.214} C_DIS
LIN {X -0.197,Y -394.552,Z 559.592,A 0.000,B 0.000,C 90.000,E1 286.622} C_DIS
LIN {X -0.155,Y -411.521,Z 559.581,A 0.000,B 0.000,C 90.000,E1 284.647} C_DIS
LIN {X 0.094,Y -423.522,Z 559.574,A 0.000,B 0.000,C 90.000,E1 283.244} C_DIS
LIN {X 0.083,Y -434.996,Z 559.566,A 0.000,B 0.000,C 90.000,E1 281.895} C_DIS
LIN {X 0.027,Y -443.711,Z 559.560,A 0.000,B 0.000,C 90.000,E1 280.838} C_DIS
LIN {X -0.013,Y -451.866,Z 559.554,A 0.000,B 0.000,C 90.000,E1 279.792} C_DIS
LIN {X -0.136,Y -461.097,Z 559.547,A 0.000,B 0.000,C 90.000,E1 278.511} C_DIS
LIN {X 0.022,Y -467.770,Z 559.542,A 0.000,B 0.000,C 90.000,E1 277.466} C_DIS
LIN {X 0.198,Y -473.699,Z 559.536,A 0.000,B 0.000,C 90.000,E1 276.429} C_DIS
LIN {X 0.117,Y -477.510,Z 559.532,A 0.000,B 0.000,C 90.000,E1 275.682} C_DIS
LIN {X -0.220,Y -479.805,Z 559.529,A 0.000,B 0.000,C 90.000,E1 275.220} C_DIS
LIN {X -0.066,Y -481.753,Z 559.526,A 0.000,B 0.000,C 90.000,E1 274.702} C_DIS
LIN {X 0.056,Y -483.409,Z 559.523,A 0.000,B 0.000,C 90.000,E1 274.188} C_DIS
LIN {X 0.227,Y -484.769,Z 559.521,A 0.000,B 0.000,C 90.000,E1 273.669} C_DIS
LIN {X -0.108,Y -485.866,Z 559.518,A 0.000,B 0.000,C 90.000,E1 273.212} C_DIS
LIN {X 0.077,Y -486.582,Z 559.515,A 0.000,B 0.000,C 90.000,E1 272.694} C_DIS
LIN {X -0.242,Y -486.917,Z 559.512,A 0.000,B 0.000,C 90.000,E1 272.236} C_DIS
LIN {X -0.053,Y -486.868,Z 559.510,A 0.000,B 0.000,C 90.000,E1 271.718} C_DIS
LIN {X 0.121,Y -486.334,Z 559.507,A 0.000,B 0.000,C 90.000,E1 271.203} C_DIS
LIN {X -0.189,Y -485.320,Z 559.504,A 0.000,B 0.000,C 90.000,E1 270.745} C_DIS
LIN {X -0.015,Y -483.817,Z 559.501,A 0.000,B 0.000,C 90.000,E1 270.229} C_DIS
LIN {X 0.151,Y -481.658,Z 559.499,A 0.000,B 0.000,C 90.000,E1 269.714} C_DIS
LIN {X -0.172,Y -478.812,Z 559.496,A 0.000,B 0.000,C 90.000,E1 269.255} C_DIS
LIN {X 0.135,Y -477.119,Z 559.494,A 0.000,B 0.000,C 90.000,E1 268.969} C_DIS
LIN {X -0.214,Y -472.945,Z 559.492,A 0.000,B 0.000,C 90.000,E1 268.511} C_DIS
LIN {X 0.079,Y -470.458,Z 559.490,A 0.000,B 0.000,C 90.000,E1 268.224} C_DIS
LIN {X -0.217,Y -464.570,Z 559.487,A 0.000,B 0.000,C 90.000,E1 267.764} C_DIS
LIN {X -0.099,Y -461.557,Z 559.486,A 0.000,B 0.000,C 90.000,E1 267.535} C_DIS
LIN {X -0.005,Y -454.815,Z 559.484,A 0.000,B 0.000,C 90.000,E1 267.135} C_DIS
LIN {X 0.230,Y -447.757,Z 559.482,A 0.000,B 0.000,C 90.000,E1 266.788} C_DIS
LIN {X 0.004,Y -440.519,Z 559.481,A 0.000,B 0.000,C 90.000,E1 266.560} C_DIS
LIN {X 0.180,Y -432.864,Z 559.480,A 0.000,B 0.000,C 90.000,E1 266.331} C_DIS
LIN {X -0.135,Y -424.464,Z 559.479,A 0.000,B 0.000,C 90.000,E1 266.216} C_DIS
LIN {X -0.109,Y -413.783,Z 559.478,A 0.000,B 0.000,C 90.000,E1 266.102} C_DIS
LIN {X 0.142,Y -408.775,Z 559.478,A 0.000,B 0.000,C 90.000,E1 266.045} C_DIS
LIN {X 0.028,Y -180.922,Z 559.478,A 0.000,B 0.000,C 90.000,E1 266.045} C_DIS
LIN {X 0.068,Y -180.868,Z 559.472,A 0.000,B 0.000,C 90.000,E1 265.008} C_DIS
LIN {X -0.029,Y -178.928,Z 559.443,A 0.000,B 0.000,C 90.000,E1 259.803} C_DIS
LIN {X 0.010,Y -175.976,Z 559.415,A 0.000,B 0.000,C 90.000,E1 254.700} C_DIS
LIN {X -0.045,Y -175.465,Z 559.410,A 0.000,B 0.000,C 90.000,E1 253.866} C_DIS
LIN {X 0.012,Y -172.215,Z 559.387,A 0.000,B 0.000,C 90.000,E1 249.571} C_DIS
LIN {X -0.010,Y -171.690,Z 559.382,A 0.000,B 0.000,C 90.000,E1 248.720} C_DIS
LIN {X -0.020,Y -167.917,Z 559.358,A 0.000,B 0.000,C 90.000,E1 244.409} C_DIS
LIN {X -0.002,Y -166.659,Z 559.348,A 0.000,B 0.000,C 90.000,E1 242.666} C_DIS
LIN {X -0.086,Y -162.643,Z 559.324,A 0.000,B 0.000,C 90.000,E1 238.329} C_DIS
LIN {X -0.023,Y -161.331,Z 559.314,A 0.000,B 0.000,C 90.000,E1 236.548} C_DIS
LIN {X 0.019,Y -157.326,Z 559.290,A 0.000,B 0.000,C 90.000,E1 232.110} C_DIS
LIN {X -0.048,Y -155.308,Z 559.275,A 0.000,B 0.000,C 90.000,E1 229.461} C_DIS
LIN {X -0.009,Y -151.665,Z 559.250,A 0.000,B 0.000,C 90.000,E1 224.960} C_DIS
LIN {X 0.035,Y -150.531,Z 559.240,A 0.000,B 0.000,C 90.000,E1 223.137} C_DIS
LIN {X -0.034,Y -147.257,Z 559.214,A 0.000,B 0.000,C 90.000,E1 218.624} C_DIS
LIN {X 0.023,Y -145.282,Z 559.194,A 0.000,B 0.000,C 90.000,E1 214.945} C_DIS
LIN {X 0.056,Y -142.384,Z 559.164,A 0.000,B 0.000,C 90.000,E1 209.411} C_DIS
LIN {X -0.021,Y -141.362,Z 559.148,A 0.000,B 0.000,C 90.000,E1 206.668} C_DIS
LIN {X -0.043,Y -139.343,Z 559.112,A 0.000,B 0.000,C 90.000,E1 200.174} C_DIS
LIN {X -0.037,Y -139.013,Z 559.102,A 0.000,B 0.000,C 90.000,E1 198.308} C_DIS
LIN {X -0.043,Y -138.341,Z 559.055,A 0.000,B 0.000,C 90.000,E1 189.905} C_DIS
LIN {X -0.023,Y -139.398,Z 559.008,A 0.000,B 0.000,C 90.000,E1 181.489} C_DIS
LIN {X 0.031,Y -141.301,Z 558.972,A 0.000,B 0.000,C 90.000,E1 174.951} C_DIS
LIN {X -0.012,Y -142.662,Z 558.957,A 0.000,B 0.000,C 90.000,E1 172.186} C_DIS
LIN {X -0.062,Y -145.008,Z 558.931,A 0.000,B 0.000,C 90.000,E1 167.589} C_DIS
LIN {X -0.073,Y -147.635,Z 558.911,A 0.000,B 0.000,C 90.000,E1 163.921} C_DIS
LIN {X 0.005,Y -150.265,Z 558.890,A 0.000,B 0.000,C 90.000,E1 160.242} C_DIS
LIN {X 0.018,Y -153.665,Z 558.870,A 0.000,B 0.000,C 90.000,E1 156.613} C_DIS
LIN {X 0.074,Y -157.080,Z 558.850,A 0.000,B 0.000,C 90.000,E1 152.999} C_DIS
LIN {X 0.013,Y -161.215,Z 558.830,A 0.000,B 0.000,C 90.000,E1 149.459} C_DIS
LIN {X -0.039,Y -163.304,Z 558.821,A 0.000,B 0.000,C 90.000,E1 147.709} C_DIS
LIN {X -0.029,Y -167.753,Z 558.801,A 0.000,B 0.000,C 90.000,E1 144.196} C_DIS
LIN {X -0.011,Y -171.569,Z 558.787,A 0.000,B 0.000,C 90.000,E1 141.582} C_DIS
LIN {X -0.076,Y -176.517,Z 558.767,A 0.000,B 0.000,C 90.000,E1 138.162} C_DIS
LIN {X 0.048,Y -180.814,Z 558.753,A 0.000,B 0.000,C 90.000,E1 135.567} C_DIS
LIN {X 0.033,Y -186.224,Z 558.734,A 0.000,B 0.000,C 90.000,E1 132.204} C_DIS
LIN {X -0.014,Y -191.324,Z 558.719,A 0.000,B 0.000,C 90.000,E1 129.439} C_DIS
LIN {X -0.093,Y -191.758,Z 558.718,A 0.000,B 0.000,C 90.000,E1 129.197} C_DIS
LIN {X 0.031,Y -289.369,Z 558.718,A 0.000,B 0.000,C 90.000,E1 129.152} C_DIS
LIN {X -0.109,Y -295.502,Z 558.716,A 0.000,B 0.000,C 90.000,E1 128.910} C_DIS
LIN {X -0.045,Y -298.394,Z 558.715,A 0.000,B 0.000,C 90.000,E1 128.624} C_DIS
LIN {X -0.130,Y -302.099,Z 558.711,A 0.000,B 0.000,C 90.000,E1 128.096} C_DIS
LIN {X 0.054,Y -303.678,Z 558.710,A 0.000,B 0.000,C 90.000,E1 127.729} C_DIS
LIN {X 0.056,Y -304.920,Z 558.708,A 0.000,B 0.000,C 90.000,E1 127.397} C_DIS
LIN {X -0.030,Y -316.731,Z 558.686,A 0.000,B 0.000,C 90.000,E1 123.499} C_DIS
LIN {X 0.156,Y -326.974,Z 558.670,A 0.000,B 0.000,C 90.000,E1 120.590} C_DIS
LIN {X 0.142,Y -338.566,Z 558.654,A 0.000,B 0.000,C 90.000,E1 117.769} C_DIS
LIN {X -0.008,Y -351.603,Z 558.639,A 0.000,B 0.000,C 90.000,E1 115.027} C_DIS
LIN {X -0.157,Y -364.504,Z 558.626,A 0.000,B 0.000,C 90.000,E1 112.642} C_DIS
LIN {X 0.079,Y -378.737,Z 558.613,A 0.000,B 0.000,C 90.000,E1 110.248} C_DIS
LIN {X 0.070,Y -394.404,Z 558.600,A 0.000,B 0.000,C 90.000,E1 107.946} C_DIS
LIN {X -0.061,Y -411.619,Z 558.587,A 0.000,B 0.000,C 90.000,E1 105.717} C_DIS
LIN {X -0.111,Y -430.509,Z 558.575,A 0.000,B 0.000,C 90.000,E1 103.536} C_DIS
LIN {X -0.173,Y -450.576,Z 558.564,A 0.000,B 0.000,C 90.000,E1 101.478} C_DIS
LIN {X 0.059,Y -471.199,Z 558.553,A 0.000,B 0.000,C 90.000,E1 99.557} C_DIS
LIN {X 0.171,Y -476.218,Z 558.551,A 0.000,B 0.000,C 90.000,E1 99.095} C_DIS
LIN {X -0.187,Y -478.034,Z 558.549,A 0.000,B 0.000,C 90.000,E1 98.916} C_DIS
LIN {X 0.154,Y -479.601,Z 558.548,A 0.000,B 0.000,C 90.000,E1 98.624} C_DIS
LIN {X -0.050,Y -480.774,Z 558.547,A 0.000,B 0.000,C 90.000,E1 98.398} C_DIS
LIN {X 0.177,Y -482.191,Z 558.544,A 0.000,B 0.000,C 90.000,E1 97.871} C_DIS
LIN {X -0.137,Y -482.574,Z 558.541,A 0.000,B 0.000,C 90.000,E1 97.409} C_DIS
LIN {X 0.037,Y -481.984,Z 558.538,A 0.000,B 0.000,C 90.000,E1 96.891} C_DIS
LIN {X 0.214,Y -480.327,Z 558.536,A 0.000,B 0.000,C 90.000,E1 96.372} C_DIS
LIN {X 0.035,Y -479.005,Z 558.534,A 0.000,B 0.000,C 90.000,E1 96.144} C_DIS
LIN {X 0.199,Y -475.298,Z 558.531,A 0.000,B 0.000,C 90.000,E1 95.625} C_DIS
LIN {X 0.124,Y -460.138,Z 558.520,A 0.000,B 0.000,C 90.000,E1 93.612} C_DIS
LIN {X 0.157,Y -449.963,Z 558.512,A 0.000,B 0.000,C 90.000,E1 92.064} C_DIS
LIN {X 0.110,Y -436.442,Z 558.498,A 0.000,B 0.000,C 90.000,E1 89.714} C_DIS
LIN {X 0.020,Y -428.617,Z 558.491,A 0.000,B 0.000,C 90.000,E1 88.396} C_DIS
LIN {X -0.144,Y -414.252,Z 558.478,A 0.000,B 0.000,C 90.000,E1 85.988} C_DIS
LIN {X -0.210,Y -400.228,Z 558.464,A 0.000,B 0.000,C 90.000,E1 83.514} C_DIS
LIN {X -0.145,Y -388.069,Z 558.451,A 0.000,B 0.000,C 90.000,E1 81.254} C_DIS
LIN {X 0.059,Y -377.448,Z 558.440,A 0.000,B 0.000,C 90.000,E1 79.218} C_DIS
LIN {X 0.083,Y -365.384,Z 558.427,A 0.000,B 0.000,C 90.000,E1 76.881} C_DIS
LIN {X 0.076,Y -356.923,Z 558.417,A 0.000,B 0.000,C 90.000,E1 75.102} C_DIS
LIN {X -0.127,Y -346.796,Z 558.404,A 0.000,B 0.000,C 90.000,E1 72.725} C_DIS
LIN {X 0.056,Y -335.455,Z 558.387,A 0.000,B 0.000,C 90.000,E1 69.625} C_DIS
LIN {X 0.163,Y -325.292,Z 558.370,A 0.000,B 0.000,C 90.000,E1 66.485} C_DIS
LIN {X 0.032,Y -317.706,Z 558.355,A 0.000,B 0.000,C 90.000,E1 63.973} C_DIS
LIN {X 0.132,Y -310.259,Z 558.341,A 0.000,B 0.000,C 90.000,E1 61.385} C_DIS
LIN {X 0.084,Y -302.941,Z 558.327,A 0.000,B 0.000,C 90.000,E1 58.791} C_DIS
LIN {X -0.056,Y -293.955,Z 558.308,A 0.000,B 0.000,C 90.000,E1 55.515} C_DIS
LIN {X -0.098,Y -287.201,Z 558.293,A 0.000,B 0.000,C 90.000,E1 52.844} C_DIS
LIN {X -0.056,Y -282.057,Z 558.282,A 0.000,B 0.000,C 90.000,E1 50.803} C_DIS
LIN {X -0.148,Y -276.567,Z 558.271,A 0.000,B 0.000,C 90.000,E1 48.771} C_DIS
LIN {X -0.145,Y -272.588,Z 558.263,A 0.000,B 0.000,C 90.000,E1 47.391} C_DIS
LIN {X -0.125,Y -267.155,Z 558.253,A 0.000,B 0.000,C 90.000,E1 45.648} C_DIS
LIN {X 0.032,Y -260.118,Z 558.242,A 0.000,B 0.000,C 90.000,E1 43.500} C_DIS
LIN {X -0.057,Y -248.619,Z 558.222,A 0.000,B 0.000,C 90.000,E1 39.930} C_DIS
LIN {X -0.030,Y -239.046,Z 558.203,A 0.000,B 0.000,C 90.000,E1 36.629} C_DIS
LIN {X 0.039,Y -229.415,Z 558.183,A 0.000,B 0.000,C 90.000,E1 32.880} C_DIS
LIN {X -0.087,Y -222.528,Z 558.166,A 0.000,B 0.000,C 90.000,E1 29.873} C_DIS
LIN {X 0.090,Y -216.447,Z 558.149,A 0.000,B 0.000,C 90.000,E1 26.744} C_DIS
LIN {X 0.015,Y -211.144,Z 558.131,A 0.000,B 0.000,C 90.000,E1 23.643} C_DIS
LIN {X 0.029,Y -206.746,Z 558.114,A 0.000,B 0.000,C 90.000,E1 20.482} C_DIS
LIN {X 0.027,Y -202.323,Z 558.092,A 0.000,B 0.000,C 90.000,E1 16.496} C_DIS
LIN {X 0.006,Y -198.948,Z 558.069,A 0.000,B 0.000,C 90.000,E1 12.479} C_DIS
LIN {X 0.090,Y -196.076,Z 558.038,A 0.000,B 0.000,C 90.000,E1 6.777} C_DIS
LIN {X 0.069,Y -195.591,Z 557.988,A 0.000,B 0.000,C 90.000,E1 357.879} C_DIS
LIN {X 0.043,Y -197.969,Z 557.957,A 0.000,B 0.000,C 90.000,E1 352.186} C_DIS
LIN {X -0.045,Y -201.437,Z 557.930,A 0.000,B 0.000,C 90.000,E1 347.353} C_DIS
LIN {X -0.076,Y -206.119,Z 557.903,A 0.000,B 0.000,C 90.000,E1 342.543} C_DIS
LIN {X 0.028,Y -210.883,Z 557.881,A 0.000,B 0.000,C 90.000,E1 338.539} C_DIS
LIN {X 0.092,Y -216.330,Z 557.859,A 0.000,B 0.000,C 90.000,E1 334.588} C_DIS
LIN {X 0.030,Y -222.355,Z 557.837,A 0.000,B 0.000,C 90.000,E1 330.717} C_DIS
LIN {X -0.105,Y -228.979,Z 557.816,A 0.000,B 0.000,C 90.000,E1 326.914} C_DIS
LIN {X -0.111,Y -236.204,Z 557.795,A 0.000,B 0.000,C 90.000,E1 323.130} C_DIS
LIN {X -0.020,Y -243.852,Z 557.774,A 0.000,B 0.000,C 90.000,E1 319.380} C_DIS
LIN {X -0.103,Y -252.386,Z 557.754,A 0.000,B 0.000,C 90.000,E1 315.729} C_DIS
LIN {X 0.057,Y -261.223,Z 557.736,A 0.000,B 0.000,C 90.000,E1 312.447} C_DIS
LIN {X 0.065,Y -272.294,Z 557.716,A 0.000,B 0.000,C 90.000,E1 308.910} C_DIS
LIN {X -0.027,Y -284.911,Z 557.697,A 0.000,B 0.000,C 90.000,E1 305.471} C_DIS
LIN {X 0.029,Y -298.931,Z 557.678,A 0.000,B 0.000,C 90.000,E1 302.084} C_DIS
LIN {X -0.106,Y -314.131,Z 557.660,A 0.000,B 0.000,C 90.000,E1 298.821} C_DIS
LIN {X -0.038,Y -328.921,Z 557.644,A 0.000,B 0.000,C 90.000,E1 295.924} C_DIS
LIN {X 0.053,Y -341.625,Z 557.632,A 0.000,B 0.000,C 90.000,E1 293.718} C_DIS
LIN {X -0.036,Y -355.777,Z 557.620,A 0.000,B 0.000,C 90.000,E1 291.589} C_DIS
LIN {X 0.070,Y -378.053,Z 557.603,A 0.000,B 0.000,C 90.000,E1 288.598} C_DIS
LIN {X -0.068,Y -396.999,Z 557.591,A 0.000,B 0.000,C 90.000,E1 286.315} C_DIS
LIN {X -0.050,Y -413.983,Z 557.580,A 0.000,B 0.000,C 90.000,E1 284.356} C_DIS
LIN {X 0.078,Y -423.559,Z 557.574,A 0.000,B 0.000,C 90.000,E1 283.244} C_DIS
LIN {X 0.069,Y -435.099,Z 557.566,A 0.000,B 0.000,C 90.000,E1 281.895} C_DIS
LIN {X 0.013,Y -443.808,Z 557.560,A 0.000,B 0.000,C 90.000,E1 280.838} C_DIS
LIN {X -0.027,Y -451.963,Z 557.554,A 0.000,B 0.000,C 90.000,E1 279.792} C_DIS
LIN {X 0.032,Y -459.419,Z 557.549,A 0.000,B 0.000,C 90.000,E1 278.746} C_DIS
LIN {X 0.177,Y -466.299,Z 557.543,A 0.000,B 0.000,C 90.000,E1 277.701} C_DIS
LIN {X 0.091,Y -470.949,Z 557.539,A 0.000,B 0.000,C 90.000,E1 276.947} C_DIS
LIN {X -0.018,Y -475.176,Z 557.534,A 0.000,B 0.000,C 90.000,E1 276.201} C_DIS
LIN {X -0.081,Y -478.803,Z 557.530,A 0.000,B 0.000,C 90.000,E1 275.454} C_DIS
LIN {X -0.074,Y -481.805,Z 557.526,A 0.000,B 0.000,C 90.000,E1 274.702} C_DIS
LIN {X 0.049,Y -483.447,Z 557.523,A 0.000,B 0.000,C 90.000,E1 274.188} C_DIS
LIN {X 0.220,Y -484.784,Z 557.521,A 0.000,B 0.000,C 90.000,E1 273.669} C_DIS
LIN {X -0.115,Y -485.835,Z 557.518,A 0.000,B 0.000,C 90.000,E1 273.212} C_DIS
LIN {X 0.070,Y -486.557,Z 557.515,A 0.000,B 0.000,C 90.000,E1 272.694} C_DIS
LIN {X 0.238,Y -486.884,Z 557.512,A 0.000,B 0.000,C 90.000,E1 272.178} C_DIS
LIN {X -0.060,Y -486.812,Z 557.510,A 0.000,B 0.000,C 90.000,E1 271.718} C_DIS
LIN {X 0.115,Y -486.310,Z 557.507,A 0.000,B 0.000,C 90.000,E1 271.203} C_DIS
LIN {X -0.195,Y -485.301,Z 557.504,A 0.000,B 0.000,C 90.000,E1 270.745} C_DIS
LIN {X -0.023,Y -483.713,Z 557.501,A 0.000,B 0.000,C 90.000,E1 270.229} C_DIS
LIN {X 0.144,Y -481.595,Z 557.498,A 0.000,B 0.000,C 90.000,E1 269.714} C_DIS
LIN {X -0.018,Y -480.348,Z 557.497,A 0.000,B 0.000,C 90.000,E1 269.484} C_DIS
LIN {X 0.127,Y -477.068,Z 557.494,A 0.000,B 0.000,C 90.000,E1 268.969} C_DIS
LIN {X -0.222,Y -472.939,Z 557.492,A 0.000,B 0.000,C 90.000,E1 268.511} C_DIS
LIN {X -0.040,Y -467.722,Z 557.489,A 0.000,B 0.000,C 90.000,E1 267.993} C_DIS
LIN {X -0.166,Y -464.671,Z 557.487,A 0.000,B 0.000,C 90.000,E1 267.764} C_DIS
LIN {X -0.049,Y -461.571,Z 557.486,A 0.000,B 0.000,C 90.000,E1 267.535} C_DIS
LIN {X 0.029,Y -454.815,Z 557.484,A 0.000,B 0.000,C 90.000,E1 267.135} C_DIS
LIN {X -0.203,Y -447.723,Z 557.482,A 0.000,B 0.000,C 90.000,E1 266.846} C_DIS
LIN {X 0.011,Y -440.548,Z 557.481,A 0.000,B 0.000,C 90.000,E1 266.560} C_DIS
LIN {X 0.187,Y -432.909,Z 557.480,A 0.000,B 0.000,C 90.000,E1 266.331} C_DIS
LIN {X -0.144,Y -424.582,Z 557.479,A 0.000,B 0.000,C 90.000,E1 266.216} C_DIS
LIN {X -0.136,Y -413.461,Z 557.478,A 0.000,B 0.000,C 90.000,E1 266.102} C_DIS
LIN {X 0.114,Y -408.259,Z 557.478,A 0.000,B 0.000,C 90.000,E1 266.045} C_DIS
LIN {X 0.016,Y -180.922,Z 557.478,A 0.000,B 0.000,C 90.000,E1 266.045} C_DIS
LIN {X 0.057,Y -180.867,Z 557.472,A 0.000,B 0.000,C 90.000,E1 265.008} C_DIS
LIN {X -0.040,Y -178.927,Z 557.443,A 0.000,B 0.000,C 90.000,E1 259.803} C_DIS
LIN {X -0.002,Y -175.974,Z 557.415,A 0.000,B 0.000,C 90.000,E1 254.700} C_DIS
LIN {X -0.057,Y -175.461,Z 557.410,A 0.000,B 0.000,C 90.000,E1 253.866} C_DIS
LIN {X 0.000,Y -172.212,Z 557.387,A 0.000,B 0.000,C 90.000,E1 249.571} C_DIS
LIN {X -0.022,Y -171.687,Z 557.382,A 0.000,B 0.000,C 90.000,E1 248.720} C_DIS
LIN {X -0.031,Y -167.914,Z 557.358,A 0.000,B 0.000,C 90.000,E1 244.409} C_DIS
LIN {X -0.013,Y -166.656,Z 557.348,A 0.000,B 0.000,C 90.000,E1 242.666} C_DIS
LIN {X 0.041,Y -162.639,Z 557.324,A 0.000,B 0.000,C 90.000,E1 238.280} C_DIS
LIN {X -0.035,Y -161.328,Z 557.314,A 0.000,B 0.000,C 90.000,E1 236.548} C_DIS
LIN {X 0.008,Y -157.323,Z 557.289,A 0.000,B 0.000,C 90.000,E1 232.110} C_DIS
LIN {X -0.059,Y -155.304,Z 557.275,A 0.000,B 0.000,C 90.000,E1 229.461} C_DIS
LIN {X -0.019,Y -151.662,Z 557.250,A 0.000,B 0.000,C 90.000,E1 224.960} C_DIS
LIN {X 0.025,Y -150.529,Z 557.240,A 0.000,B 0.000,C 90.000,E1 223.137} C_DIS
LIN {X -0.044,Y -147.254,Z 557.214,A 0.000,B 0.000,C 90.000,E1 218.624} C_DIS
LIN {X 0.012,Y -145.280,Z 557.194,A 0.000,B 0.000,C 90.000,E1 214.945} C_DIS
LIN {X 0.046,Y -142.383,Z 557.164,A 0.000,B 0.000,C 90.000,E1 209.411} C_DIS
LIN {X -0.031,Y -141.360,Z 557.148,A 0.000,B 0.000,C 90.000,E1 206.668} C_DIS
LIN {X -0.053,Y -139.342,Z 557.112,A 0.000,B 0.000,C 90.000,E1 200.174} C_DIS
LIN {X -0.048,Y -139.012,Z 557.102,A 0.000,B 0.000,C 90.000,E1 198.308} C_DIS
LIN {X -0.053,Y -138.341,Z 557.055,A 0.000,B 0.000,C 90.000,E1 189.905} C_DIS
LIN {X -0.033,Y -139.399,Z 557.008,A 0.000,B 0.000,C 90.000,E1 181.489} C_DIS
LIN {X 0.021,Y -141.302,Z 556.972,A 0.000,B 0.000,C 90.000,E1 174.951} C_DIS
LIN {X -0.022,Y -142.664,Z 556.957,A 0.000,B 0.000,C 90.000,E1 172.186} C_DIS
LIN {X -0.072,Y -145.010,Z 556.931,A 0.000,B 0.000,C 90.000,E1 167.589} C_DIS
LIN {X 0.059,Y -147.637,Z 556.910,A 0.000,B 0.000,C 90.000,E1 163.866} C_DIS
LIN {X -0.006,Y -150.268,Z 556.890,A 0.000,B 0.000,C 90.000,E1 160.242} C_DIS
LIN {X 0.008,Y -153.669,Z 556.870,A 0.000,B 0.000,C 90.000,E1 156.613} C_DIS
LIN {X 0.064,Y -157.084,Z 556.850,A 0.000,B 0.000,C 90.000,E1 152.999} C_DIS
LIN {X 0.002,Y -161.220,Z 556.830,A 0.000,B 0.000,C 90.000,E1 149.459} C_DIS
LIN {X -0.050,Y -163.309,Z 556.820,A 0.000,B 0.000,C 90.000,E1 147.709} C_DIS
LIN {X -0.040,Y -167.758,Z 556.801,A 0.000,B 0.000,C 90.000,E1 144.196} C_DIS
LIN {X -0.023,Y -171.574,Z 556.786,A 0.000,B 0.000,C 90.000,E1 141.582} C_DIS
LIN {X -0.088,Y -176.522,Z 556.767,A 0.000,B 0.000,C 90.000,E1 138.162} C_DIS
LIN {X 0.036,Y -180.821,Z 556.753,A 0.000,B 0.000,C 90.000,E1 135.567} C_DIS
LIN {X 0.022,Y -186.230,Z 556.734,A 0.000,B 0.000,C 90.000,E1 132.204} C_DIS
LIN {X -0.027,Y -191.331,Z 556.719,A 0.000,B 0.000,C 90.000,E1 129.439} C_DIS
LIN {X 0.007,Y -191.782,Z 556.718,A 0.000,B 0.000,C 90.000,E1 129.152} C_DIS
LIN {X 0.146,Y -289.083,Z 556.717,A 0.000,B 0.000,C 90.000,E1 129.116} C_DIS
LIN {X 0.010,Y -290.628,Z 556.717,A 0.000,B 0.000,C 90.000,E1 129.116} C_DIS
LIN {X -0.128,Y -295.354,Z 556.716,A 0.000,B 0.000,C 90.000,E1 128.910} C_DIS
LIN {X -0.041,Y -298.576,Z 556.714,A 0.000,B 0.000,C 90.000,E1 128.588} C_DIS
LIN {X 0.111,Y -302.221,Z 556.711,A 0.000,B 0.000,C 90.000,E1 128.016} C_DIS
LIN {X -0.130,Y -303.778,Z 556.709,A 0.000,B 0.000,C 90.000,E1 127.729} C_DIS
LIN {X 0.057,Y -305.004,Z 556.708,A 0.000,B 0.000,C 90.000,E1 127.363} C_DIS
LIN {X 0.047,Y -316.823,Z 556.686,A 0.000,B 0.000,C 90.000,E1 123.452} C_DIS
LIN {X -0.035,Y -327.081,Z 556.670,A 0.000,B 0.000,C 90.000,E1 120.590} C_DIS
LIN {X -0.053,Y -338.689,Z 556.654,A 0.000,B 0.000,C 90.000,E1 117.769} C_DIS
LIN {X -0.207,Y -351.743,Z 556.639,A 0.000,B 0.000,C 90.000,E1 115.027} C_DIS
LIN {X -0.024,Y -364.661,Z 556.625,A 0.000,B 0.000,C 90.000,E1 112.589} C_DIS
LIN {X -0.127,Y -378.911,Z 556.612,A 0.000,B 0.000,C 90.000,E1 110.248} C_DIS
LIN {X -0.139,Y -394.597,Z 556.600,A 0.000,B 0.000,C 90.000,E1 107.946} C_DIS
LIN {X 0.121,Y -411.835,Z 556.587,A 0.000,B 0.000,C 90.000,E1 105.662} C_DIS
LIN {X 0.090,Y -430.746,Z 556.575,A 0.000,B 0.000,C 90.000,E1 103.480} C_DIS
LIN {X 0.059,Y -450.822,Z 556.563,A 0.000,B 0.000,C 90.000,E1 101.422} C_DIS
LIN {X -0.143,Y -471.451,Z 556.553,A 0.000,B 0.000,C 90.000,E1 99.557} C_DIS
LIN {X -0.028,Y -476.444,Z 556.551,A 0.000,B 0.000,C 90.000,E1 99.095} C_DIS
LIN {X 0.087,Y -478.237,Z 556.549,A 0.000,B 0.000,C 90.000,E1 98.859} C_DIS
LIN {X -0.044,Y -479.784,Z 556.548,A 0.000,B 0.000,C 90.000,E1 98.624} C_DIS
LIN {X -0.248,Y -480.942,Z 556.547,A 0.000,B 0.000,C 90.000,E1 98.398} C_DIS
LIN {X -0.021,Y -482.334,Z 556.544,A 0.000,B 0.000,C 90.000,E1 97.871} C_DIS
LIN {X 0.145,Y -482.692,Z 556.541,A 0.000,B 0.000,C 90.000,E1 97.352} C_DIS
LIN {X -0.159,Y -482.078,Z 556.538,A 0.000,B 0.000,C 90.000,E1 96.891} C_DIS
LIN {X 0.019,Y -480.393,Z 556.535,A 0.000,B 0.000,C 90.000,E1 96.372} C_DIS
LIN {X -0.158,Y -479.054,Z 556.534,A 0.000,B 0.000,C 90.000,E1 96.144} C_DIS
LIN {X -0.128,Y -473.367,Z 556.530,A 0.000,B 0.000,C 90.000,E1 95.391} C_DIS
LIN {X -0.061,Y -460.144,Z 556.520,A 0.000,B 0.000,C 90.000,E1 93.612} C_DIS
LIN {X -0.024,Y -449.949,Z 556.511,A 0.000,B 0.000,C 90.000,E1 92.064} C_DIS
LIN {X -0.066,Y -436.406,Z 556.498,A 0.000,B 0.000,C 90.000,E1 89.714} C_DIS
LIN {X -0.154,Y -428.565,Z 556.491,A 0.000,B 0.000,C 90.000,E1 88.396} C_DIS
LIN {X 0.131,Y -414.202,Z 556.477,A 0.000,B 0.000,C 90.000,E1 85.927} C_DIS
LIN {X -0.016,Y -401.698,Z 556.465,A 0.000,B 0.000,C 90.000,E1 83.742} C_DIS
LIN {X 0.026,Y -389.496,Z 556.453,A 0.000,B 0.000,C 90.000,E1 81.489} C_DIS
LIN {X -0.153,Y -380.381,Z 556.443,A 0.000,B 0.000,C 90.000,E1 79.803} C_DIS
LIN {X -0.049,Y -369.761,Z 556.432,A 0.000,B 0.000,C 90.000,E1 77.757} C_DIS
LIN {X -0.090,Y -359.503,Z 556.420,A 0.000,B 0.000,C 90.000,E1 75.700} C_DIS
LIN {X 0.127,Y -347.875,Z 556.405,A 0.000,B 0.000,C 90.000,E1 72.960} C_DIS
LIN {X -0.087,Y -337.512,Z 556.390,A 0.000,B 0.000,C 90.000,E1 70.242} C_DIS
LIN {X 0.080,Y -327.197,Z 556.373,A 0.000,B 0.000,C 90.000,E1 67.102} C_DIS
LIN {X 0.023,Y -317.630,Z 556.355,A 0.000,B 0.000,C 90.000,E1 63.948} C_DIS
LIN {X -0.015,Y -310.193,Z 556.341,A 0.000,B 0.000,C 90.000,E1 61.385} C_DIS
LIN {X -0.061,Y -302.870,Z 556.327,A 0.000,B 0.000,C 90.000,E1 58.791} C_DIS
LIN {X 0.044,Y -293.879,Z 556.308,A 0.000,B 0.000,C 90.000,E1 55.468} C_DIS
LIN {X 0.162,Y -287.099,Z 556.293,A 0.000,B 0.000,C 90.000,E1 52.763} C_DIS
LIN {X 0.021,Y -281.950,Z 556.282,A 0.000,B 0.000,C 90.000,E1 50.759} C_DIS
LIN {X 0.102,Y -276.464,Z 556.271,A 0.000,B 0.000,C 90.000,E1 48.690} C_DIS
LIN {X 0.101,Y -272.445,Z 556.263,A 0.000,B 0.000,C 90.000,E1 47.310} C_DIS
LIN {X 0.114,Y -266.986,Z 556.253,A 0.000,B 0.000,C 90.000,E1 45.567} C_DIS
LIN {X 0.073,Y -259.928,Z 556.242,A 0.000,B 0.000,C 90.000,E1 43.461} C_DIS
LIN {X -0.019,Y -249.556,Z 556.224,A 0.000,B 0.000,C 90.000,E1 40.253} C_DIS
LIN {X 0.035,Y -240.921,Z 556.207,A 0.000,B 0.000,C 90.000,E1 37.317} C_DIS
LIN {X 0.125,Y -232.987,Z 556.191,A 0.000,B 0.000,C 90.000,E1 34.326} C_DIS
LIN {X 0.008,Y -225.689,Z 556.174,A 0.000,B 0.000,C 90.000,E1 31.337} C_DIS
LIN {X -0.016,Y -219.227,Z 556.157,A 0.000,B 0.000,C 90.000,E1 28.281} C_DIS
LIN {X 0.068,Y -213.580,Z 556.140,A 0.000,B 0.000,C 90.000,E1 25.155} C_DIS
LIN {X 0.030,Y -208.737,Z 556.122,A 0.000,B 0.000,C 90.000,E1 22.025} C_DIS
LIN {X 0.031,Y -203.899,Z 556.100,A 0.000,B 0.000,C 90.000,E1 18.055} C_DIS
LIN {X -0.040,Y -200.071,Z 556.078,A 0.000,B 0.000,C 90.000,E1 14.064} C_DIS
LIN {X -0.034,Y -196.636,Z 556.047,A 0.000,B 0.000,C 90.000,E1 8.398} C_DIS
LIN {X -0.083,Y -195.391,Z 555.993,A 0.000,B 0.000,C 90.000,E1 358.740} C_DIS
LIN {X 0.042,Y -197.945,Z 555.957,A 0.000,B 0.000,C 90.000,E1 352.186} C_DIS
LIN {X -0.048,Y -201.407,Z 555.930,A 0.000,B 0.000,C 90.000,E1 347.353} C_DIS
LIN {X -0.080,Y -206.091,Z 555.903,A 0.000,B 0.000,C 90.000,E1 342.543} C_DIS
LIN {X 0.023,Y -210.858,Z 555.881,A 0.000,B 0.000,C 90.000,E1 338.539} C_DIS
LIN {X 0.085,Y -216.312,Z 555.859,A 0.000,B 0.000,C 90.000,E1 334.588} C_DIS
LIN {X 0.024,Y -222.323,Z 555.837,A 0.000,B 0.000,C 90.000,E1 330.717} C_DIS
LIN {X -0.113,Y -228.937,Z 555.816,A 0.000,B 0.000,C 90.000,E1 326.914} C_DIS
LIN {X -0.121,Y -236.174,Z 555.795,A 0.000,B 0.000,C 90.000,E1 323.130} C_DIS
LIN {X -0.031,Y -243.821,Z 555.774,A 0.000,B 0.000,C 90.000,E1 319.380} C_DIS
LIN {X -0.116,Y -252.392,Z 555.754,A 0.000,B 0.000,C 90.000,E1 315.729} C_DIS
LIN {X 0.044,Y -261.223,Z 555.736,A 0.000,B 0.000,C 90.000,E1 312.447} C_DIS
LIN {X 0.052,Y -272.295,Z 555.716,A 0.000,B 0.000,C 90.000,E1 308.910} C_DIS
LIN {X -0.042,Y -284.908,Z 555.697,A 0.000,B 0.000,C 90.000,E1 305.471} C_DIS
LIN {X 0.013,Y -298.899,Z 555.678,A 0.000,B 0.000,C 90.000,E1 302.084} C_DIS
LIN {X -0.124,Y -314.079,Z 555.660,A 0.000,B 0.000,C 90.000,E1 298.821} C_DIS
LIN {X -0.005,Y -327.116,Z 555.646,A 0.000,B 0.000,C 90.000,E1 296.232} C_DIS
LIN {X 0.167,Y -341.561,Z 555.632,A 0.000,B 0.000,C 90.000,E1 293.695} C_DIS
LIN {X -0.062,Y -355.743,Z 555.620,A 0.000,B 0.000,C 90.000,E1 291.589} C_DIS
LIN {X -0.154,Y -373.429,Z 555.607,A 0.000,B 0.000,C 90.000,E1 289.214} C_DIS
LIN {X 0.083,Y -392.218,Z 555.594,A 0.000,B 0.000,C 90.000,E1 286.858} C_DIS
LIN {X -0.012,Y -409.166,Z 555.583,A 0.000,B 0.000,C 90.000,E1 284.898} C_DIS
LIN {X -0.116,Y -421.296,Z 555.575,A 0.000,B 0.000,C 90.000,E1 283.536} C_DIS
LIN {X 0.011,Y -432.846,Z 555.568,A 0.000,B 0.000,C 90.000,E1 282.175} C_DIS
LIN {X -0.165,Y -441.734,Z 555.562,A 0.000,B 0.000,C 90.000,E1 281.130} C_DIS
LIN {X -0.153,Y -450.043,Z 555.556,A 0.000,B 0.000,C 90.000,E1 280.074} C_DIS
LIN {X -0.127,Y -457.683,Z 555.550,A 0.000,B 0.000,C 90.000,E1 279.029} C_DIS
LIN {X -0.076,Y -464.721,Z 555.544,A 0.000,B 0.000,C 90.000,E1 277.992} C_DIS
LIN {X -0.181,Y -469.555,Z 555.540,A 0.000,B 0.000,C 90.000,E1 277.239} C_DIS
LIN {X 0.020,Y -475.248,Z 555.534,A 0.000,B 0.000,C 90.000,E1 276.201} C_DIS
LIN {X -0.043,Y -478.834,Z 555.530,A 0.000,B 0.000,C 90.000,E1 275.454} C_DIS
LIN {X -0.035,Y -481.848,Z 555.526,A 0.000,B 0.000,C 90.000,E1 274.702} C_DIS
LIN {X 0.087,Y -483.469,Z 555.523,A 0.000,B 0.000,C 90.000,E1 274.188} C_DIS
LIN {X -0.224,Y -484.790,Z 555.521,A 0.000,B 0.000,C 90.000,E1 273.726} C_DIS
LIN {X -0.075,Y -485.832,Z 555.518,A 0.000,B 0.000,C 90.000,E1 273.212} C_DIS
LIN {X 0.110,Y -486.513,Z 555.515,A 0.000,B 0.000,C 90.000,E1 272.694} C_DIS
LIN {X -0.209,Y -486.836,Z 555.512,A 0.000,B 0.000,C 90.000,E1 272.236} C_DIS
LIN {X -0.020,Y -486.760,Z 555.510,A 0.000,B 0.000,C 90.000,E1 271.718} C_DIS
LIN {X 0.153,Y -486.231,Z 555.507,A 0.000,B 0.000,C 90.000,E1 271.203} C_DIS
LIN {X -0.157,Y -485.260,Z 555.504,A 0.000,B 0.000,C 90.000,E1 270.745} C_DIS
LIN {X 0.015,Y -483.687,Z 555.501,A 0.000,B 0.000,C 90.000,E1 270.229} C_DIS
LIN {X 0.182,Y -481.581,Z 555.499,A 0.000,B 0.000,C 90.000,E1 269.714} C_DIS
LIN {X -0.142,Y -478.794,Z 555.496,A 0.000,B 0.000,C 90.000,E1 269.255} C_DIS
LIN {X -0.007,Y -475.163,Z 555.493,A 0.000,B 0.000,C 90.000,E1 268.740} C_DIS
LIN {X 0.107,Y -470.490,Z 555.490,A 0.000,B 0.000,C 90.000,E1 268.224} C_DIS
LIN {X -0.040,Y -467.710,Z 555.489,A 0.000,B 0.000,C 90.000,E1 267.993} C_DIS
LIN {X -0.200,Y -464.600,Z 555.487,A 0.000,B 0.000,C 90.000,E1 267.764} C_DIS
LIN {X 0.032,Y -457.938,Z 555.485,A 0.000,B 0.000,C 90.000,E1 267.306} C_DIS
LIN {X -0.027,Y -450.987,Z 555.483,A 0.000,B 0.000,C 90.000,E1 266.963} C_DIS
LIN {X -0.002,Y -443.859,Z 555.482,A 0.000,B 0.000,C 90.000,E1 266.674} C_DIS
LIN {X -0.064,Y -436.189,Z 555.480,A 0.000,B 0.000,C 90.000,E1 266.445} C_DIS
LIN {X -0.106,Y -428.525,Z 555.479,A 0.000,B 0.000,C 90.000,E1 266.274} C_DIS
LIN {X 0.161,Y -418.954,Z 555.478,A 0.000,B 0.000,C 90.000,E1 266.102} C_DIS
LIN {X 0.089,Y -407.820,Z 555.478,A 0.000,B 0.000,C 90.000,E1 266.045} C_DIS
LIN {X 0.005,Y -180.922,Z 555.478,A 0.000,B 0.000,C 90.000,E1 266.045} C_DIS
LIN {X 0.046,Y -180.867,Z 555.472,A 0.000,B 0.000,C 90.000,E1 265.008} C_DIS
LIN {X -0.051,Y -178.925,Z 555.443,A 0.000,B 0.000,C 90.000,E1 259.803} C_DIS
LIN {X -0.013,Y -175.973,Z 555.415,A 0.000,B 0.000,C 90.000,E1 254.700} C_DIS
LIN {X -0.068,Y -175.458,Z 555.410,A 0.000,B 0.000,C 90.000,E1 253.866} C_DIS
LIN {X -0.011,Y -172.209,Z 555.386,A 0.000,B 0.000,C 90.000,E1 249.571} C_DIS
LIN {X -0.033,Y -171.685,Z 555.382,A 0.000,B 0.000,C 90.000,E1 248.720} C_DIS
LIN {X -0.042,Y -167.912,Z 555.358,A 0.000,B 0.000,C 90.000,E1 244.409} C_DIS
LIN {X -0.023,Y -166.652,Z 555.348,A 0.000,B 0.000,C 90.000,E1 242.666} C_DIS
LIN {X 0.031,Y -162.636,Z 555.324,A 0.000,B 0.000,C 90.000,E1 238.280} C_DIS
LIN {X -0.045,Y -161.325,Z 555.314,A 0.000,B 0.000,C 90.000,E1 236.548} C_DIS
LIN {X -0.001,Y -157.320,Z 555.289,A 0.000,B 0.000,C 90.000,E1 232.110} C_DIS
LIN {X -0.068,Y -155.300,Z 555.275,A 0.000,B 0.000,C 90.000,E1 229.461} C_DIS
LIN {X 0.078,Y -151.660,Z 555.250,A 0.000,B 0.000,C 90.000,E1 224.919} C_DIS
LIN {X 0.015,Y -150.527,Z 555.240,A 0.000,B 0.000,C 90.000,E1 223.137} C_DIS
LIN {X -0.054,Y -147.251,Z 555.214,A 0.000,B 0.000,C 90.000,E1 218.624} C_DIS
LIN {X 0.002,Y -145.276,Z 555.194,A 0.000,B 0.000,C 90.000,E1 214.945} C_DIS
LIN {X 0.036,Y -142.381,Z 555.163,A 0.000,B 0.000,C 90.000,E1 209.411} C_DIS
LIN {X -0.041,Y -141.359,Z 555.148,A 0.000,B 0.000,C 90.000,E1 206.668} C_DIS
LIN {X 0.068,Y -139.342,Z 555.112,A 0.000,B 0.000,C 90.000,E1 200.120} C_DIS
LIN {X -0.014,Y -139.010,Z 555.102,A 0.000,B 0.000,C 90.000,E1 198.290} C_DIS
LIN {X -0.062,Y -138.340,Z 555.055,A 0.000,B 0.000,C 90.000,E1 189.905} C_DIS
LIN {X -0.042,Y -139.400,Z 555.008,A 0.000,B 0.000,C 90.000,E1 181.489} C_DIS
LIN {X 0.011,Y -141.304,Z 554.972,A 0.000,B 0.000,C 90.000,E1 174.951} C_DIS
LIN {X -0.031,Y -142.665,Z 554.957,A 0.000,B 0.000,C 90.000,E1 172.186} C_DIS
LIN {X -0.082,Y -145.012,Z 554.931,A 0.000,B 0.000,C 90.000,E1 167.589} C_DIS
LIN {X 0.048,Y -147.640,Z 554.910,A 0.000,B 0.000,C 90.000,E1 163.866} C_DIS
LIN {X -0.015,Y -150.272,Z 554.890,A 0.000,B 0.000,C 90.000,E1 160.242} C_DIS
LIN {X -0.002,Y -153.673,Z 554.870,A 0.000,B 0.000,C 90.000,E1 156.613} C_DIS
LIN {X 0.054,Y -157.088,Z 554.850,A 0.000,B 0.000,C 90.000,E1 152.999} C_DIS
LIN {X -0.008,Y -161.224,Z 554.830,A 0.000,B 0.000,C 90.000,E1 149.459} C_DIS
LIN {X 0.078,Y -163.313,Z 554.820,A 0.000,B 0.000,C 90.000,E1 147.661} C_DIS
LIN {X -0.051,Y -167.764,Z 554.801,A 0.000,B 0.000,C 90.000,E1 144.196} C_DIS
LIN {X 0.101,Y -171.579,Z 554.786,A 0.000,B 0.000,C 90.000,E1 141.537} C_DIS
LIN {X -0.099,Y -176.528,Z 554.767,A 0.000,B 0.000,C 90.000,E1 138.162} C_DIS
LIN {X 0.025,Y -180.827,Z 554.753,A 0.000,B 0.000,C 90.000,E1 135.567} C_DIS
LIN {X 0.009,Y -186.236,Z 554.734,A 0.000,B 0.000,C 90.000,E1 132.204} C_DIS
LIN {X -0.039,Y -191.336,Z 554.719,A 0.000,B 0.000,C 90.000,E1 129.439} C_DIS
LIN {X 0.084,Y -191.803,Z 554.717,A 0.000,B 0.000,C 90.000,E1 129.116} C_DIS
LIN {X 0.081,Y -288.514,Z 554.717,A 0.000,B 0.000,C 90.000,E1 129.116} C_DIS
LIN {X -0.010,Y -290.058,Z 554.717,A 0.000,B 0.000,C 90.000,E1 129.116} C_DIS
LIN {X -0.145,Y -295.195,Z 554.716,A 0.000,B 0.000,C 90.000,E1 128.910} C_DIS
LIN {X 0.066,Y -298.276,Z 554.714,A 0.000,B 0.000,C 90.000,E1 128.588} C_DIS
LIN {X -0.123,Y -301.960,Z 554.711,A 0.000,B 0.000,C 90.000,E1 128.096} C_DIS
LIN {X 0.061,Y -303.582,Z 554.710,A 0.000,B 0.000,C 90.000,E1 127.729} C_DIS
LIN {X 0.061,Y -304.855,Z 554.708,A 0.000,B 0.000,C 90.000,E1 127.397} C_DIS
LIN {X -0.026,Y -316.687,Z 554.686,A 0.000,B 0.000,C 90.000,E1 123.499} C_DIS
LIN {X 0.159,Y -326.930,Z 554.670,A 0.000,B 0.000,C 90.000,E1 120.590} C_DIS
LIN {X 0.143,Y -338.521,Z 554.654,A 0.000,B 0.000,C 90.000,E1 117.769} C_DIS
LIN {X -0.008,Y -351.557,Z 554.639,A 0.000,B 0.000,C 90.000,E1 115.027} C_DIS
LIN {X -0.158,Y -364.457,Z 554.626,A 0.000,B 0.000,C 90.000,E1 112.642} C_DIS
LIN {X 0.076,Y -378.689,Z 554.613,A 0.000,B 0.000,C 90.000,E1 110.248} C_DIS
LIN {X 0.067,Y -394.355,Z 554.600,A 0.000,B 0.000,C 90.000,E1 107.946} C_DIS
LIN {X -0.065,Y -411.571,Z 554.587,A 0.000,B 0.000,C 90.000,E1 105.717} C_DIS
LIN {X -0.117,Y -430.460,Z 554.575,A 0.000,B 0.000,C 90.000,E1 103.536} C_DIS
LIN {X -0.181,Y -450.529,Z 554.564,A 0.000,B 0.000,C 90.000,E1 101.478} C_DIS
LIN {X 0.050,Y -471.151,Z 554.553,A 0.000,B 0.000,C 90.000,E1 99.557} C_DIS
LIN {X 0.162,Y -476.227,Z 554.551,A 0.000,B 0.000,C 90.000,E1 99.095} C_DIS
LIN {X -0.197,Y -478.098,Z 554.549,A 0.000,B 0.000,C 90.000,E1 98.916} C_DIS
LIN {X 0.144,Y -479.709,Z 554.548,A 0.000,B 0.000,C 90.000,E1 98.624} C_DIS
LIN {X -0.060,Y -480.915,Z 554.547,A 0.000,B 0.000,C 90.000,E1 98.398} C_DIS
LIN {X 0.167,Y -482.382,Z 554.544,A 0.000,B 0.000,C 90.000,E1 97.871} C_DIS
LIN {X -0.145,Y -482.807,Z 554.541,A 0.000,B 0.000,C 90.000,E1 97.409} C_DIS
LIN {X 0.030,Y -482.260,Z 554.538,A 0.000,B 0.000,C 90.000,E1 96.891} C_DIS
LIN {X 0.207,Y -480.654,Z 554.536,A 0.000,B 0.000,C 90.000,E1 96.372} C_DIS
LIN {X 0.030,Y -479.367,Z 554.534,A 0.000,B 0.000,C 90.000,E1 96.144} C_DIS
LIN {X 0.197,Y -475.701,Z 554.531,A 0.000,B 0.000,C 90.000,E1 95.625} C_DIS
LIN {X 0.130,Y -460.475,Z 554.520,A 0.000,B 0.000,C 90.000,E1 93.612} C_DIS
LIN {X 0.167,Y -450.222,Z 554.512,A 0.000,B 0.000,C 90.000,E1 92.064} C_DIS
LIN {X 0.126,Y -436.636,Z 554.498,A 0.000,B 0.000,C 90.000,E1 89.714} C_DIS
LIN {X 0.039,Y -428.800,Z 554.491,A 0.000,B 0.000,C 90.000,E1 88.396} C_DIS
LIN {X -0.120,Y -414.433,Z 554.478,A 0.000,B 0.000,C 90.000,E1 85.988} C_DIS
LIN {X 0.175,Y -401.916,Z 554.465,A 0.000,B 0.000,C 90.000,E1 83.742} C_DIS
LIN {X -0.169,Y -389.694,Z 554.453,A 0.000,B 0.000,C 90.000,E1 81.546} C_DIS
LIN {X 0.063,Y -379.035,Z 554.442,A 0.000,B 0.000,C 90.000,E1 79.511} C_DIS
LIN {X 0.125,Y -366.886,Z 554.429,A 0.000,B 0.000,C 90.000,E1 77.173} C_DIS
LIN {X 0.054,Y -358.256,Z 554.419,A 0.000,B 0.000,C 90.000,E1 75.408} C_DIS
LIN {X -0.099,Y -346.777,Z 554.404,A 0.000,B 0.000,C 90.000,E1 72.725} C_DIS
LIN {X -0.033,Y -335.480,Z 554.387,A 0.000,B 0.000,C 90.000,E1 69.645} C_DIS
LIN {X -0.108,Y -325.332,Z 554.370,A 0.000,B 0.000,C 90.000,E1 66.538} C_DIS
LIN {X 0.066,Y -315.854,Z 554.352,A 0.000,B 0.000,C 90.000,E1 63.332} C_DIS
LIN {X -0.151,Y -308.446,Z 554.338,A 0.000,B 0.000,C 90.000,E1 60.795} C_DIS
LIN {X 0.175,Y -301.083,Z 554.323,A 0.000,B 0.000,C 90.000,E1 58.122} C_DIS
LIN {X -0.031,Y -292.247,Z 554.305,A 0.000,B 0.000,C 90.000,E1 54.848} C_DIS
LIN {X 0.043,Y -285.476,Z 554.290,A 0.000,B 0.000,C 90.000,E1 52.145} C_DIS
LIN {X 0.007,Y -280.243,Z 554.278,A 0.000,B 0.000,C 90.000,E1 50.114} C_DIS
LIN {X -0.125,Y -276.508,Z 554.271,A 0.000,B 0.000,C 90.000,E1 48.771} C_DIS
LIN {X -0.122,Y -272.477,Z 554.263,A 0.000,B 0.000,C 90.000,E1 47.391} C_DIS
LIN {X -0.104,Y -267.023,Z 554.253,A 0.000,B 0.000,C 90.000,E1 45.648} C_DIS
LIN {X 0.001,Y -261.159,Z 554.244,A 0.000,B 0.000,C 90.000,E1 43.866} C_DIS
LIN {X 0.108,Y -250.701,Z 554.226,A 0.000,B 0.000,C 90.000,E1 40.620} C_DIS
LIN {X -0.011,Y -240.940,Z 554.208,A 0.000,B 0.000,C 90.000,E1 37.363} C_DIS
LIN {X -0.058,Y -232.984,Z 554.191,A 0.000,B 0.000,C 90.000,E1 34.405} C_DIS
LIN {X -0.048,Y -225.677,Z 554.174,A 0.000,B 0.000,C 90.000,E1 31.386} C_DIS
LIN {X 0.011,Y -219.219,Z 554.157,A 0.000,B 0.000,C 90.000,E1 28.309} C_DIS
LIN {X 0.003,Y -213.582,Z 554.140,A 0.000,B 0.000,C 90.000,E1 25.207} C_DIS
LIN {X -0.037,Y -208.748,Z 554.123,A 0.000,B 0.000,C 90.000,E1 22.078} C_DIS
LIN {X -0.040,Y -203.883,Z 554.101,A 0.000,B 0.000,C 90.000,E1 18.109} C_DIS
LIN {X 0.080,Y -200.048,Z 554.078,A 0.000,B 0.000,C 90.000,E1 14.064} C_DIS
LIN {X 0.082,Y -196.613,Z 554.047,A 0.000,B 0.000,C 90.000,E1 8.398} C_DIS
LIN {X -0.084,Y -195.353,Z 553.993,A 0.000,B 0.000,C 90.000,E1 358.740} C_DIS
LIN {X 0.040,Y -197.913,Z 553.957,A 0.000,B 0.000,C 90.000,E1 352.186} C_DIS
LIN {X -0.051,Y -201.372,Z 553.930,A 0.000,B 0.000,C 90.000,E1 347.353} C_DIS
LIN {X -0.084,Y -206.054,Z 553.903,A 0.000,B 0.000,C 90.000,E1 342.543} C_DIS
LIN {X 0.017,Y -210.823,Z 553.881,A 0.000,B 0.000,C 90.000,E1 338.539} C_DIS
LIN {X 0.078,Y -216.283,Z 553.859,A 0.000,B 0.000,C 90.000,E1 334.588} C_DIS
LIN {X -0.070,Y -221.053,Z 553.842,A 0.000,B 0.000,C 90.000,E1 331.513} C_DIS
LIN {X -0.057,Y -227.512,Z 553.820,A 0.000,B 0.000,C 90.000,E1 327.661} C_DIS
LIN {X 0.086,Y -234.644,Z 553.799,A 0.000,B 0.000,C 90.000,E1 323.829} C_DIS
LIN {X -0.125,Y -240.642,Z 553.783,A 0.000,B 0.000,C 90.000,E1 320.884} C_DIS
LIN {X 0.053,Y -248.813,Z 553.762,A 0.000,B 0.000,C 90.000,E1 317.148} C_DIS
LIN {X -0.063,Y -258.142,Z 553.742,A 0.000,B 0.000,C 90.000,E1 313.542} C_DIS
LIN {X 0.009,Y -268.840,Z 553.722,A 0.000,B 0.000,C 90.000,E1 309.967} C_DIS
LIN {X 0.037,Y -279.685,Z 553.705,A 0.000,B 0.000,C 90.000,E1 306.824} C_DIS
LIN {X 0.011,Y -293.114,Z 553.686,A 0.000,B 0.000,C 90.000,E1 303.420} C_DIS
LIN {X 0.102,Y -307.852,Z 553.667,A 0.000,B 0.000,C 90.000,E1 300.079} C_DIS
LIN {X -0.057,Y -323.661,Z 553.649,A 0.000,B 0.000,C 90.000,E1 296.873} C_DIS
LIN {X 0.044,Y -335.919,Z 553.637,A 0.000,B 0.000,C 90.000,E1 294.643} C_DIS
LIN {X 0.136,Y -347.444,Z 553.627,A 0.000,B 0.000,C 90.000,E1 292.770} C_DIS
LIN {X -0.028,Y -364.369,Z 553.613,A 0.000,B 0.000,C 90.000,E1 290.375} C_DIS
LIN {X 0.108,Y -382.741,Z 553.600,A 0.000,B 0.000,C 90.000,E1 288.000} C_DIS
LIN {X -0.078,Y -399.504,Z 553.589,A 0.000,B 0.000,C 90.000,E1 286.024} C_DIS
LIN {X -0.002,Y -416.550,Z 553.578,A 0.000,B 0.000,C 90.000,E1 284.064} C_DIS
LIN {X -0.022,Y -428.407,Z 553.571,A 0.000,B 0.000,C 90.000,E1 282.703} C_DIS
LIN {X -0.253,Y -437.551,Z 553.565,A 0.000,B 0.000,C 90.000,E1 281.658} C_DIS
LIN {X 0.151,Y -446.151,Z 553.559,A 0.000,B 0.000,C 90.000,E1 280.546} C_DIS
LIN {X 0.141,Y -454.142,Z 553.553,A 0.000,B 0.000,C 90.000,E1 279.500} C_DIS
LIN {X -0.230,Y -461.495,Z 553.547,A 0.000,B 0.000,C 90.000,E1 278.511} C_DIS
LIN {X -0.069,Y -468.195,Z 553.541,A 0.000,B 0.000,C 90.000,E1 277.466} C_DIS
LIN {X -0.206,Y -472.683,Z 553.537,A 0.000,B 0.000,C 90.000,E1 276.720} C_DIS
LIN {X 0.230,Y -476.616,Z 553.533,A 0.000,B 0.000,C 90.000,E1 275.910} C_DIS
LIN {X 0.175,Y -480.044,Z 553.529,A 0.000,B 0.000,C 90.000,E1 275.163} C_DIS
LIN {X -0.149,Y -481.973,Z 553.526,A 0.000,B 0.000,C 90.000,E1 274.702} C_DIS
LIN {X -0.025,Y -483.551,Z 553.523,A 0.000,B 0.000,C 90.000,E1 274.188} C_DIS
LIN {X 0.147,Y -484.848,Z 553.521,A 0.000,B 0.000,C 90.000,E1 273.669} C_DIS
LIN {X -0.188,Y -485.815,Z 553.518,A 0.000,B 0.000,C 90.000,E1 273.212} C_DIS
LIN {X -0.002,Y -486.472,Z 553.515,A 0.000,B 0.000,C 90.000,E1 272.694} C_DIS
LIN {X 0.166,Y -486.799,Z 553.512,A 0.000,B 0.000,C 90.000,E1 272.178} C_DIS
LIN {X -0.132,Y -486.696,Z 553.509,A 0.000,B 0.000,C 90.000,E1 271.718} C_DIS
LIN {X 0.042,Y -486.175,Z 553.507,A 0.000,B 0.000,C 90.000,E1 271.203} C_DIS
LIN {X 0.216,Y -485.151,Z 553.504,A 0.000,B 0.000,C 90.000,E1 270.688} C_DIS
LIN {X -0.098,Y -483.641,Z 553.501,A 0.000,B 0.000,C 90.000,E1 270.229} C_DIS
LIN {X 0.068,Y -481.496,Z 553.498,A 0.000,B 0.000,C 90.000,E1 269.714} C_DIS
LIN {X 0.224,Y -478.679,Z 553.496,A 0.000,B 0.000,C 90.000,E1 269.198} C_DIS
LIN {X -0.119,Y -475.021,Z 553.493,A 0.000,B 0.000,C 90.000,E1 268.740} C_DIS
LIN {X 0.175,Y -472.812,Z 553.492,A 0.000,B 0.000,C 90.000,E1 268.453} C_DIS
LIN {X -0.131,Y -467.559,Z 553.489,A 0.000,B 0.000,C 90.000,E1 267.993} C_DIS
LIN {X 0.193,Y -464.434,Z 553.487,A 0.000,B 0.000,C 90.000,E1 267.707} C_DIS
LIN {X -0.135,Y -461.363,Z 553.486,A 0.000,B 0.000,C 90.000,E1 267.535} C_DIS
LIN {X -0.006,Y -454.609,Z 553.484,A 0.000,B 0.000,C 90.000,E1 267.135} C_DIS
LIN {X -0.198,Y -447.720,Z 553.482,A 0.000,B 0.000,C 90.000,E1 266.846} C_DIS
LIN {X 0.016,Y -440.580,Z 553.481,A 0.000,B 0.000,C 90.000,E1 266.560} C_DIS
LIN {X 0.184,Y -433.077,Z 553.480,A 0.000,B 0.000,C 90.000,E1 266.331} C_DIS
LIN {X -0.137,Y -424.888,Z 553.479,A 0.000,B 0.000,C 90.000,E1 266.216} C_DIS
LIN {X -0.131,Y -414.757,Z 553.478,A 0.000,B 0.000,C 90.000,E1 266.102} C_DIS
LIN {X 0.031,Y -405.537,Z 553.478,A 0.000,B 0.000,C 90.000,E1 266.045} C_DIS
LIN {X -0.004,Y -180.922,Z 553.478,A 0.000,B 0.000,C 90.000,E1 266.045} C_DIS
LIN {X 0.054,Y -180.867,Z 553.472,A 0.000,B 0.000,C 90.000,E1 265.008} C_DIS
LIN {X -0.043,Y -178.927,Z 553.443,A 0.000,B 0.000,C 90.000,E1 259.803} C_DIS
LIN {X -0.005,Y -175.973,Z 553.415,A 0.000,B 0.000,C 90.000,E1 254.700} C_DIS
LIN {X -0.060,Y -175.460,Z 553.410,A 0.000,B 0.000,C 90.000,E1 253.866} C_DIS
LIN {X -0.002,Y -172.212,Z 553.386,A 0.000,B 0.000,C 90.000,E1 249.571} C_DIS
LIN {X -0.025,Y -171.687,Z 553.382,A 0.000,B 0.000,C 90.000,E1 248.720} C_DIS
LIN {X -0.034,Y -167.913,Z 553.358,A 0.000,B 0.000,C 90.000,E1 244.409} C_DIS
LIN {X -0.015,Y -166.655,Z 553.348,A 0.000,B 0.000,C 90.000,E1 242.666} C_DIS
LIN {X 0.038,Y -162.639,Z 553.324,A 0.000,B 0.000,C 90.000,E1 238.280} C_DIS
LIN {X -0.037,Y -161.327,Z 553.314,A 0.000,B 0.000,C 90.000,E1 236.548} C_DIS
LIN {X 0.006,Y -157.322,Z 553.289,A 0.000,B 0.000,C 90.000,E1 232.110} C_DIS
LIN {X -0.061,Y -155.303,Z 553.275,A 0.000,B 0.000,C 90.000,E1 229.461} C_DIS
LIN {X -0.022,Y -151.661,Z 553.250,A 0.000,B 0.000,C 90.000,E1 224.960} C_DIS
LIN {X 0.022,Y -150.528,Z 553.240,A 0.000,B 0.000,C 90.000,E1 223.137} C_DIS
LIN {X -0.047,Y -147.253,Z 553.214,A 0.000,B 0.000,C 90.000,E1 218.624} C_DIS
LIN {X 0.009,Y -145.279,Z 553.194,A 0.000,B 0.000,C 90.000,E1 214.945} C_DIS
LIN {X 0.043,Y -142.382,Z 553.164,A 0.000,B 0.000,C 90.000,E1 209.411} C_DIS
LIN {X -0.035,Y -141.359,Z 553.148,A 0.000,B 0.000,C 90.000,E1 206.668} C_DIS
LIN {X 0.075,Y -139.342,Z 553.112,A 0.000,B 0.000,C 90.000,E1 200.120} C_DIS
LIN {X -0.050,Y -139.011,Z 553.102,A 0.000,B 0.000,C 90.000,E1 198.308} C_DIS
LIN {X -0.055,Y -138.341,Z 553.055,A 0.000,B 0.000,C 90.000,E1 189.905} C_DIS
LIN {X -0.035,Y -139.399,Z 553.008,A 0.000,B 0.000,C 90.000,E1 181.489} C_DIS
LIN {X 0.018,Y -141.304,Z 552.972,A 0.000,B 0.000,C 90.000,E1 174.951} C_DIS
LIN {X -0.025,Y -142.664,Z 552.957,A 0.000,B 0.000,C 90.000,E1 172.186} C_DIS
LIN {X -0.075,Y -145.011,Z 552.931,A 0.000,B 0.000,C 90.000,E1 167.589} C_DIS
LIN {X 0.056,Y -147.637,Z 552.910,A 0.000,B 0.000,C 90.000,E1 163.866} C_DIS
LIN {X -0.008,Y -150.269,Z 552.890,A 0.000,B 0.000,C 90.000,E1 160.242} C_DIS
LIN {X 0.005,Y -153.670,Z 552.870,A 0.000,B 0.000,C 90.000,E1 156.613} C_DIS
LIN {X 0.061,Y -157.085,Z 552.850,A 0.000,B 0.000,C 90.000,E1 152.999} C_DIS
LIN {X 0.000,Y -161.221,Z 552.830,A 0.000,B 0.000,C 90.000,E1 149.459} C_DIS
LIN {X -0.053,Y -163.310,Z 552.820,A 0.000,B 0.000,C 90.000,E1 147.709} C_DIS
LIN {X -0.043,Y -167.759,Z 552.801,A 0.000,B 0.000,C 90.000,E1 144.196} C_DIS
LIN {X 0.109,Y -171.575,Z 552.786,A 0.000,B 0.000,C 90.000,E1 141.537} C_DIS
LIN {X -0.092,Y -176.524,Z 552.767,A 0.000,B 0.000,C 90.000,E1 138.162} C_DIS
LIN {X 0.033,Y -180.823,Z 552.753,A 0.000,B 0.000,C 90.000,E1 135.567} C_DIS
LIN {X 0.018,Y -186.232,Z 552.734,A 0.000,B 0.000,C 90.000,E1 132.204} C_DIS
LIN {X -0.033,Y -191.333,Z 552.719,A 0.000,B 0.000,C 90.000,E1 129.439} C_DIS
LIN {X 0.029,Y -191.830,Z 552.717,A 0.000,B 0.000,C 90.000,E1 129.116} C_DIS
LIN {X -0.002,Y -288.238,Z 552.717,A 0.000,B 0.000,C 90.000,E1 129.116} C_DIS
LIN {X 0.047,Y -292.967,Z 552.717,A 0.000,B 0.000,C 90.000,E1 128.991} C_DIS
LIN {X -0.132,Y -294.942,Z 552.716,A 0.000,B 0.000,C 90.000,E1 128.910} C_DIS
LIN {X -0.089,Y -298.799,Z 552.714,A 0.000,B 0.000,C 90.000,E1 128.543} C_DIS
LIN {X -0.133,Y -302.336,Z 552.711,A 0.000,B 0.000,C 90.000,E1 128.016} C_DIS
LIN {X 0.053,Y -303.881,Z 552.709,A 0.000,B 0.000,C 90.000,E1 127.649} C_DIS
LIN {X 0.055,Y -305.095,Z 552.707,A 0.000,B 0.000,C 90.000,E1 127.317} C_DIS
LIN {X 0.175,Y -315.867,Z 552.687,A 0.000,B 0.000,C 90.000,E1 123.706} C_DIS
LIN {X -0.108,Y -326.004,Z 552.671,A 0.000,B 0.000,C 90.000,E1 120.875} C_DIS
LIN {X 0.013,Y -337.474,Z 552.656,A 0.000,B 0.000,C 90.000,E1 118.025} C_DIS
LIN {X -0.178,Y -350.389,Z 552.640,A 0.000,B 0.000,C 90.000,E1 115.283} C_DIS
LIN {X 0.114,Y -363.170,Z 552.627,A 0.000,B 0.000,C 90.000,E1 112.823} C_DIS
LIN {X -0.030,Y -377.272,Z 552.614,A 0.000,B 0.000,C 90.000,E1 110.482} C_DIS
LIN {X -0.087,Y -392.800,Z 552.601,A 0.000,B 0.000,C 90.000,E1 108.181} C_DIS
LIN {X 0.127,Y -409.865,Z 552.588,A 0.000,B 0.000,C 90.000,E1 105.898} C_DIS
LIN {X 0.042,Y -428.593,Z 552.576,A 0.000,B 0.000,C 90.000,E1 103.716} C_DIS
LIN {X -0.143,Y -448.606,Z 552.565,A 0.000,B 0.000,C 90.000,E1 101.658} C_DIS
LIN {X 0.049,Y -469.179,Z 552.554,A 0.000,B 0.000,C 90.000,E1 99.726} C_DIS
LIN {X 0.128,Y -474.402,Z 552.552,A 0.000,B 0.000,C 90.000,E1 99.265} C_DIS
LIN {X 0.247,Y -476.744,Z 552.550,A 0.000,B 0.000,C 90.000,E1 99.029} C_DIS
LIN {X -0.182,Y -478.519,Z 552.549,A 0.000,B 0.000,C 90.000,E1 98.859} C_DIS
LIN {X 0.160,Y -480.053,Z 552.548,A 0.000,B 0.000,C 90.000,E1 98.568} C_DIS
LIN {X -0.041,Y -481.201,Z 552.546,A 0.000,B 0.000,C 90.000,E1 98.341} C_DIS
LIN {X 0.188,Y -482.577,Z 552.544,A 0.000,B 0.000,C 90.000,E1 97.814} C_DIS
LIN {X -0.122,Y -482.922,Z 552.541,A 0.000,B 0.000,C 90.000,E1 97.352} C_DIS
LIN {X 0.055,Y -482.294,Z 552.538,A 0.000,B 0.000,C 90.000,E1 96.834} C_DIS
LIN {X 0.234,Y -480.591,Z 552.535,A 0.000,B 0.000,C 90.000,E1 96.315} C_DIS
LIN {X 0.056,Y -479.240,Z 552.534,A 0.000,B 0.000,C 90.000,E1 96.087} C_DIS
LIN {X 0.086,Y -473.523,Z 552.530,A 0.000,B 0.000,C 90.000,E1 95.334} C_DIS
LIN {X 0.151,Y -460.254,Z 552.520,A 0.000,B 0.000,C 90.000,E1 93.555} C_DIS
LIN {X 0.187,Y -450.011,Z 552.511,A 0.000,B 0.000,C 90.000,E1 92.007} C_DIS
LIN {X -0.034,Y -437.937,Z 552.500,A 0.000,B 0.000,C 90.000,E1 89.943} C_DIS
LIN {X -0.095,Y -430.153,Z 552.492,A 0.000,B 0.000,C 90.000,E1 88.625} C_DIS
LIN {X 0.101,Y -417.331,Z 552.480,A 0.000,B 0.000,C 90.000,E1 86.445} C_DIS
LIN {X -0.038,Y -406.321,Z 552.470,A 0.000,B 0.000,C 90.000,E1 84.546} C_DIS
LIN {X 0.069,Y -393.998,Z 552.457,A 0.000,B 0.000,C 90.000,E1 82.299} C_DIS
LIN {X -0.053,Y -383.324,Z 552.446,A 0.000,B 0.000,C 90.000,E1 80.330} C_DIS
LIN {X 0.106,Y -372.624,Z 552.435,A 0.000,B 0.000,C 90.000,E1 78.285} C_DIS
LIN {X 0.058,Y -359.330,Z 552.420,A 0.000,B 0.000,C 90.000,E1 75.644} C_DIS
LIN {X -0.071,Y -347.727,Z 552.405,A 0.000,B 0.000,C 90.000,E1 72.960} C_DIS
LIN {X 0.024,Y -335.274,Z 552.387,A 0.000,B 0.000,C 90.000,E1 69.571} C_DIS
LIN {X -0.179,Y -325.146,Z 552.369,A 0.000,B 0.000,C 90.000,E1 66.485} C_DIS
LIN {X 0.120,Y -317.524,Z 552.355,A 0.000,B 0.000,C 90.000,E1 63.896} C_DIS
LIN {X -0.202,Y -310.094,Z 552.341,A 0.000,B 0.000,C 90.000,E1 61.385} C_DIS
LIN {X 0.013,Y -302.702,Z 552.326,A 0.000,B 0.000,C 90.000,E1 58.742} C_DIS
LIN {X -0.140,Y -293.773,Z 552.308,A 0.000,B 0.000,C 90.000,E1 55.468} C_DIS
LIN {X -0.021,Y -286.964,Z 552.293,A 0.000,B 0.000,C 90.000,E1 52.763} C_DIS
LIN {X 0.017,Y -281.826,Z 552.282,A 0.000,B 0.000,C 90.000,E1 50.723} C_DIS
LIN {X -0.080,Y -276.271,Z 552.270,A 0.000,B 0.000,C 90.000,E1 48.690} C_DIS
LIN {X -0.079,Y -272.206,Z 552.263,A 0.000,B 0.000,C 90.000,E1 47.310} C_DIS
LIN {X -0.066,Y -266.708,Z 552.253,A 0.000,B 0.000,C 90.000,E1 45.567} C_DIS
LIN {X -0.109,Y -259.621,Z 552.241,A 0.000,B 0.000,C 90.000,E1 43.461} C_DIS
LIN {X -0.041,Y -249.267,Z 552.223,A 0.000,B 0.000,C 90.000,E1 40.216} C_DIS
LIN {X -0.002,Y -240.640,Z 552.207,A 0.000,B 0.000,C 90.000,E1 37.282} C_DIS
LIN {X -0.059,Y -232.681,Z 552.191,A 0.000,B 0.000,C 90.000,E1 34.326} C_DIS
LIN {X 0.132,Y -225.408,Z 552.174,A 0.000,B 0.000,C 90.000,E1 31.258} C_DIS
LIN {X -0.011,Y -218.980,Z 552.157,A 0.000,B 0.000,C 90.000,E1 28.231} C_DIS
LIN {X -0.121,Y -213.372,Z 552.140,A 0.000,B 0.000,C 90.000,E1 25.155} C_DIS
LIN {X 0.035,Y -208.590,Z 552.122,A 0.000,B 0.000,C 90.000,E1 21.972} C_DIS
LIN {X 0.035,Y -203.727,Z 552.100,A 0.000,B 0.000,C 90.000,E1 18.000} C_DIS
LIN {X -0.036,Y -199.928,Z 552.078,A 0.000,B 0.000,C 90.000,E1 14.008} C_DIS
LIN {X -0.033,Y -196.532,Z 552.046,A 0.000,B 0.000,C 90.000,E1 8.341} C_DIS
LIN {X 0.068,Y -195.495,Z 551.988,A 0.000,B 0.000,C 90.000,E1 357.879} C_DIS
LIN {X 0.030,Y -198.362,Z 551.952,A 0.000,B 0.000,C 90.000,E1 351.376} C_DIS
LIN {X 0.040,Y -202.031,Z 551.925,A 0.000,B 0.000,C 90.000,E1 346.520} C_DIS
LIN {X 0.037,Y -206.906,Z 551.898,A 0.000,B 0.000,C 90.000,E1 341.710} C_DIS
LIN {X 0.036,Y -211.843,Z 551.876,A 0.000,B 0.000,C 90.000,E1 337.741} C_DIS
LIN {X 0.023,Y -217.399,Z 551.855,A 0.000,B 0.000,C 90.000,E1 333.819} C_DIS
LIN {X -0.011,Y -223.501,Z 551.833,A 0.000,B 0.000,C 90.000,E1 329.950} C_DIS
LIN {X -0.066,Y -230.263,Z 551.812,A 0.000,B 0.000,C 90.000,E1 326.135} C_DIS
LIN {X -0.144,Y -236.088,Z 551.795,A 0.000,B 0.000,C 90.000,E1 323.130} C_DIS
LIN {X -0.059,Y -243.736,Z 551.774,A 0.000,B 0.000,C 90.000,E1 319.380} C_DIS
LIN {X -0.148,Y -252.365,Z 551.754,A 0.000,B 0.000,C 90.000,E1 315.729} C_DIS
LIN {X 0.046,Y -262.250,Z 551.734,A 0.000,B 0.000,C 90.000,E1 312.081} C_DIS
LIN {X 0.093,Y -273.494,Z 551.714,A 0.000,B 0.000,C 90.000,E1 308.543} C_DIS
LIN {X 0.037,Y -286.219,Z 551.695,A 0.000,B 0.000,C 90.000,E1 305.105} C_DIS
LIN {X -0.029,Y -300.297,Z 551.676,A 0.000,B 0.000,C 90.000,E1 301.750} C_DIS
LIN {X -0.074,Y -312.406,Z 551.662,A 0.000,B 0.000,C 90.000,E1 299.127} C_DIS
LIN {X -0.059,Y -326.987,Z 551.646,A 0.000,B 0.000,C 90.000,E1 296.232} C_DIS
LIN {X -0.023,Y -339.596,Z 551.633,A 0.000,B 0.000,C 90.000,E1 294.027} C_DIS
LIN {X 0.143,Y -351.494,Z 551.623,A 0.000,B 0.000,C 90.000,E1 292.153} C_DIS
LIN {X 0.167,Y -371.105,Z 551.608,A 0.000,B 0.000,C 90.000,E1 289.450} C_DIS
LIN {X -0.155,Y -387.491,Z 551.597,A 0.000,B 0.000,C 90.000,E1 287.457} C_DIS
LIN {X 0.135,Y -404.441,Z 551.586,A 0.000,B 0.000,C 90.000,E1 285.426} C_DIS
LIN {X 0.071,Y -419.041,Z 551.577,A 0.000,B 0.000,C 90.000,E1 283.772} C_DIS
LIN {X 0.084,Y -430.868,Z 551.569,A 0.000,B 0.000,C 90.000,E1 282.411} C_DIS
LIN {X -0.113,Y -439.866,Z 551.563,A 0.000,B 0.000,C 90.000,E1 281.366} C_DIS
LIN {X -0.120,Y -448.334,Z 551.557,A 0.000,B 0.000,C 90.000,E1 280.310} C_DIS
LIN {X -0.110,Y -456.187,Z 551.551,A 0.000,B 0.000,C 90.000,E1 279.265} C_DIS
LIN {X -0.008,Y -463.392,Z 551.546,A 0.000,B 0.000,C 90.000,E1 278.219} C_DIS
LIN {X -0.122,Y -468.348,Z 551.541,A 0.000,B 0.000,C 90.000,E1 277.466} C_DIS
LIN {X 0.213,Y -472.821,Z 551.537,A 0.000,B 0.000,C 90.000,E1 276.663} C_DIS
LIN {X 0.179,Y -476.758,Z 551.533,A 0.000,B 0.000,C 90.000,E1 275.910} C_DIS
LIN {X 0.126,Y -480.149,Z 551.529,A 0.000,B 0.000,C 90.000,E1 275.163} C_DIS
LIN {X -0.199,Y -482.024,Z 551.526,A 0.000,B 0.000,C 90.000,E1 274.702} C_DIS
LIN {X -0.074,Y -483.595,Z 551.523,A 0.000,B 0.000,C 90.000,E1 274.188} C_DIS
LIN {X 0.097,Y -484.881,Z 551.520,A 0.000,B 0.000,C 90.000,E1 273.669} C_DIS
LIN {X -0.236,Y -485.826,Z 551.518,A 0.000,B 0.000,C 90.000,E1 273.212} C_DIS
LIN {X -0.051,Y -486.421,Z 551.515,A 0.000,B 0.000,C 90.000,E1 272.694} C_DIS
LIN {X 0.116,Y -486.733,Z 551.512,A 0.000,B 0.000,C 90.000,E1 272.178} C_DIS
LIN {X -0.181,Y -486.630,Z 551.509,A 0.000,B 0.000,C 90.000,E1 271.718} C_DIS
LIN {X -0.009,Y -486.090,Z 551.507,A 0.000,B 0.000,C 90.000,E1 271.203} C_DIS
LIN {X 0.165,Y -485.096,Z 551.504,A 0.000,B 0.000,C 90.000,E1 270.688} C_DIS
LIN {X -0.147,Y -483.588,Z 551.501,A 0.000,B 0.000,C 90.000,E1 270.229} C_DIS
LIN {X 0.018,Y -481.450,Z 551.498,A 0.000,B 0.000,C 90.000,E1 269.714} C_DIS
LIN {X 0.174,Y -478.598,Z 551.496,A 0.000,B 0.000,C 90.000,E1 269.198} C_DIS
LIN {X -0.169,Y -474.934,Z 551.493,A 0.000,B 0.000,C 90.000,E1 268.740} C_DIS
LIN {X 0.125,Y -472.720,Z 551.492,A 0.000,B 0.000,C 90.000,E1 268.453} C_DIS
LIN {X -0.181,Y -467.449,Z 551.489,A 0.000,B 0.000,C 90.000,E1 267.993} C_DIS
LIN {X -0.172,Y -461.267,Z 551.486,A 0.000,B 0.000,C 90.000,E1 267.535} C_DIS
LIN {X -0.035,Y -454.505,Z 551.484,A 0.000,B 0.000,C 90.000,E1 267.135} C_DIS
LIN {X 0.208,Y -447.564,Z 551.482,A 0.000,B 0.000,C 90.000,E1 266.788} C_DIS
LIN {X -0.038,Y -440.354,Z 551.481,A 0.000,B 0.000,C 90.000,E1 266.560} C_DIS
LIN {X 0.126,Y -432.758,Z 551.480,A 0.000,B 0.000,C 90.000,E1 266.331} C_DIS
LIN {X -0.186,Y -424.569,Z 551.479,A 0.000,B 0.000,C 90.000,E1 266.216} C_DIS
LIN {X -0.172,Y -414.473,Z 551.478,A 0.000,B 0.000,C 90.000,E1 266.102} C_DIS
LIN {X 0.075,Y -410.086,Z 551.478,A 0.000,B 0.000,C 90.000,E1 266.045} C_DIS
LIN {X -0.003,Y -180.922,Z 551.478,A 0.000,B 0.000,C 90.000,E1 266.045} C_DIS
LIN {X 0.037,Y -180.866,Z 551.472,A 0.000,B 0.000,C 90.000,E1 265.008} C_DIS
LIN {X -0.061,Y -178.925,Z 551.443,A 0.000,B 0.000,C 90.000,E1 259.803} C_DIS
LIN {X -0.022,Y -175.971,Z 551.415,A 0.000,B 0.000,C 90.000,E1 254.700} C_DIS
LIN {X -0.028,Y -175.456,Z 551.410,A 0.000,B 0.000,C 90.000,E1 253.850} C_DIS
LIN {X -0.019,Y -172.208,Z 551.386,A 0.000,B 0.000,C 90.000,E1 249.571} C_DIS
LIN {X -0.041,Y -171.683,Z 551.382,A 0.000,B 0.000,C 90.000,E1 248.720} C_DIS
LIN {X -0.050,Y -167.909,Z 551.358,A 0.000,B 0.000,C 90.000,E1 244.409} C_DIS
LIN {X -0.032,Y -166.650,Z 551.348,A 0.000,B 0.000,C 90.000,E1 242.666} C_DIS
LIN {X 0.023,Y -162.634,Z 551.324,A 0.000,B 0.000,C 90.000,E1 238.280} C_DIS
LIN {X 0.082,Y -161.322,Z 551.314,A 0.000,B 0.000,C 90.000,E1 236.501} C_DIS
LIN {X -0.009,Y -157.318,Z 551.289,A 0.000,B 0.000,C 90.000,E1 232.110} C_DIS
LIN {X -0.077,Y -155.298,Z 551.275,A 0.000,B 0.000,C 90.000,E1 229.461} C_DIS
LIN {X 0.070,Y -151.657,Z 551.250,A 0.000,B 0.000,C 90.000,E1 224.919} C_DIS
LIN {X 0.007,Y -150.525,Z 551.240,A 0.000,B 0.000,C 90.000,E1 223.137} C_DIS
LIN {X 0.030,Y -147.250,Z 551.214,A 0.000,B 0.000,C 90.000,E1 218.588} C_DIS
LIN {X -0.005,Y -145.275,Z 551.194,A 0.000,B 0.000,C 90.000,E1 214.945} C_DIS
LIN {X 0.029,Y -142.380,Z 551.163,A 0.000,B 0.000,C 90.000,E1 209.411} C_DIS
LIN {X -0.049,Y -141.357,Z 551.148,A 0.000,B 0.000,C 90.000,E1 206.668} C_DIS
LIN {X 0.061,Y -139.341,Z 551.112,A 0.000,B 0.000,C 90.000,E1 200.120} C_DIS
LIN {X -0.021,Y -139.009,Z 551.102,A 0.000,B 0.000,C 90.000,E1 198.290} C_DIS
LIN {X -0.069,Y -138.340,Z 551.055,A 0.000,B 0.000,C 90.000,E1 189.905} C_DIS
LIN {X -0.050,Y -139.401,Z 551.008,A 0.000,B 0.000,C 90.000,E1 181.489} C_DIS
LIN {X 0.003,Y -141.306,Z 550.972,A 0.000,B 0.000,C 90.000,E1 174.951} C_DIS
LIN {X -0.039,Y -142.667,Z 550.956,A 0.000,B 0.000,C 90.000,E1 172.186} C_DIS
LIN {X 0.083,Y -145.015,Z 550.931,A 0.000,B 0.000,C 90.000,E1 167.521} C_DIS
LIN {X 0.041,Y -147.642,Z 550.910,A 0.000,B 0.000,C 90.000,E1 163.866} C_DIS
LIN {X -0.024,Y -150.274,Z 550.890,A 0.000,B 0.000,C 90.000,E1 160.242} C_DIS
LIN {X -0.011,Y -153.676,Z 550.870,A 0.000,B 0.000,C 90.000,E1 156.613} C_DIS
LIN {X 0.045,Y -157.091,Z 550.850,A 0.000,B 0.000,C 90.000,E1 152.999} C_DIS
LIN {X -0.016,Y -161.228,Z 550.830,A 0.000,B 0.000,C 90.000,E1 149.459} C_DIS
LIN {X 0.069,Y -163.316,Z 550.820,A 0.000,B 0.000,C 90.000,E1 147.661} C_DIS
LIN {X -0.060,Y -167.767,Z 550.801,A 0.000,B 0.000,C 90.000,E1 144.196} C_DIS
LIN {X 0.092,Y -171.583,Z 550.786,A 0.000,B 0.000,C 90.000,E1 141.537} C_DIS
LIN {X -0.108,Y -176.533,Z 550.767,A 0.000,B 0.000,C 90.000,E1 138.162} C_DIS
LIN {X 0.016,Y -180.831,Z 550.753,A 0.000,B 0.000,C 90.000,E1 135.567} C_DIS
LIN {X 0.001,Y -186.241,Z 550.734,A 0.000,B 0.000,C 90.000,E1 132.204} C_DIS
LIN {X -0.051,Y -191.342,Z 550.719,A 0.000,B 0.000,C 90.000,E1 129.439} C_DIS
LIN {X -0.047,Y -191.868,Z 550.717,A 0.000,B 0.000,C 90.000,E1 129.116} C_DIS
LIN {X -0.110,Y -288.959,Z 550.717,A 0.000,B 0.000,C 90.000,E1 129.116} C_DIS
LIN {X 0.035,Y -290.108,Z 550.717,A 0.000,B 0.000,C 90.000,E1 129.072} C_DIS
LIN {X -0.159,Y -294.777,Z 550.716,A 0.000,B 0.000,C 90.000,E1 128.910} C_DIS
LIN {X -0.059,Y -297.891,Z 550.715,A 0.000,B 0.000,C 90.000,E1 128.624} C_DIS
LIN {X 0.082,Y -301.589,Z 550.712,A 0.000,B 0.000,C 90.000,E1 128.096} C_DIS
LIN {X -0.159,Y -303.305,Z 550.710,A 0.000,B 0.000,C 90.000,E1 127.810} C_DIS
LIN {X 0.025,Y -304.652,Z 550.708,A 0.000,B 0.000,C 90.000,E1 127.443} C_DIS
LIN {X 0.052,Y -312.380,Z 550.693,A 0.000,B 0.000,C 90.000,E1 124.818} C_DIS
LIN {X 0.089,Y -323.194,Z 550.676,A 0.000,B 0.000,C 90.000,E1 121.592} C_DIS
LIN {X 0.129,Y -334.306,Z 550.660,A 0.000,B 0.000,C 90.000,E1 118.743} C_DIS
LIN {X 0.005,Y -346.830,Z 550.644,A 0.000,B 0.000,C 90.000,E1 115.976} C_DIS
LIN {X -0.118,Y -359.238,Z 550.631,A 0.000,B 0.000,C 90.000,E1 113.567} C_DIS
LIN {X 0.113,Y -372.940,Z 550.618,A 0.000,B 0.000,C 90.000,E1 111.153} C_DIS
LIN {X -0.049,Y -388.034,Z 550.605,A 0.000,B 0.000,C 90.000,E1 108.852} C_DIS
LIN {X 0.053,Y -404.632,Z 550.592,A 0.000,B 0.000,C 90.000,E1 106.567} C_DIS
LIN {X 0.056,Y -422.857,Z 550.580,A 0.000,B 0.000,C 90.000,E1 104.356} C_DIS
LIN {X -0.058,Y -442.613,Z 550.568,A 0.000,B 0.000,C 90.000,E1 102.243} C_DIS
LIN {X 0.194,Y -463.029,Z 550.557,A 0.000,B 0.000,C 90.000,E1 100.254} C_DIS
LIN {X -0.109,Y -475.970,Z 550.551,A 0.000,B 0.000,C 90.000,E1 99.151} C_DIS
LIN {X 0.001,Y -477.963,Z 550.550,A 0.000,B 0.000,C 90.000,E1 98.916} C_DIS
LIN {X -0.132,Y -479.667,Z 550.548,A 0.000,B 0.000,C 90.000,E1 98.681} C_DIS
LIN {X 0.138,Y -480.947,Z 550.547,A 0.000,B 0.000,C 90.000,E1 98.398} C_DIS
LIN {X -0.179,Y -482.529,Z 550.544,A 0.000,B 0.000,C 90.000,E1 97.936} C_DIS
LIN {X 0.054,Y -483.053,Z 550.541,A 0.000,B 0.000,C 90.000,E1 97.409} C_DIS
LIN {X 0.229,Y -482.603,Z 550.538,A 0.000,B 0.000,C 90.000,E1 96.891} C_DIS
LIN {X -0.070,Y -481.110,Z 550.536,A 0.000,B 0.000,C 90.000,E1 96.429} C_DIS
LIN {X -0.247,Y -479.894,Z 550.534,A 0.000,B 0.000,C 90.000,E1 96.201} C_DIS
LIN {X 0.105,Y -478.272,Z 550.533,A 0.000,B 0.000,C 90.000,E1 95.910} C_DIS
LIN {X -0.122,Y -460.987,Z 550.520,A 0.000,B 0.000,C 90.000,E1 93.669} C_DIS
LIN {X -0.071,Y -450.654,Z 550.512,A 0.000,B 0.000,C 90.000,E1 92.121} C_DIS
LIN {X -0.095,Y -437.002,Z 550.499,A 0.000,B 0.000,C 90.000,E1 89.771} C_DIS
LIN {X -0.173,Y -429.116,Z 550.491,A 0.000,B 0.000,C 90.000,E1 88.453} C_DIS
LIN {X -0.001,Y -416.335,Z 550.479,A 0.000,B 0.000,C 90.000,E1 86.274} C_DIS
LIN {X -0.102,Y -403.788,Z 550.467,A 0.000,B 0.000,C 90.000,E1 84.090} C_DIS
LIN {X -0.013,Y -391.485,Z 550.455,A 0.000,B 0.000,C 90.000,E1 81.837} C_DIS
LIN {X -0.157,Y -382.303,Z 550.445,A 0.000,B 0.000,C 90.000,E1 80.151} C_DIS
LIN {X -0.083,Y -371.583,Z 550.434,A 0.000,B 0.000,C 90.000,E1 78.117} C_DIS
LIN {X -0.078,Y -358.398,Z 550.419,A 0.000,B 0.000,C 90.000,E1 75.463} C_DIS
LIN {X 0.112,Y -346.918,Z 550.404,A 0.000,B 0.000,C 90.000,E1 72.725} C_DIS
LIN {X -0.139,Y -335.643,Z 550.387,A 0.000,B 0.000,C 90.000,E1 69.699} C_DIS
LIN {X 0.099,Y -325.497,Z 550.370,A 0.000,B 0.000,C 90.000,E1 66.538} C_DIS
LIN {X -0.012,Y -315.952,Z 550.352,A 0.000,B 0.000,C 90.000,E1 63.384} C_DIS
LIN {X 0.051,Y -308.542,Z 550.338,A 0.000,B 0.000,C 90.000,E1 60.795} C_DIS
LIN {X -0.039,Y -301.146,Z 550.323,A 0.000,B 0.000,C 90.000,E1 58.201} C_DIS
LIN {X -0.073,Y -292.312,Z 550.305,A 0.000,B 0.000,C 90.000,E1 54.895} C_DIS
LIN {X 0.011,Y -285.522,Z 550.290,A 0.000,B 0.000,C 90.000,E1 52.190} C_DIS
LIN {X 0.159,Y -282.103,Z 550.282,A 0.000,B 0.000,C 90.000,E1 50.803} C_DIS
LIN {X 0.063,Y -276.532,Z 550.271,A 0.000,B 0.000,C 90.000,E1 48.771} C_DIS
LIN {X 0.065,Y -272.472,Z 550.263,A 0.000,B 0.000,C 90.000,E1 47.391} C_DIS
LIN {X 0.078,Y -266.992,Z 550.254,A 0.000,B 0.000,C 90.000,E1 45.648} C_DIS
LIN {X 0.038,Y -259.917,Z 550.242,A 0.000,B 0.000,C 90.000,E1 43.542} C_DIS
LIN {X -0.053,Y -249.536,Z 550.224,A 0.000,B 0.000,C 90.000,E1 40.334} C_DIS
LIN {X 0.005,Y -240.889,Z 550.208,A 0.000,B 0.000,C 90.000,E1 37.397} C_DIS
LIN {X 0.098,Y -232.881,Z 550.191,A 0.000,B 0.000,C 90.000,E1 34.405} C_DIS
LIN {X -0.018,Y -225.602,Z 550.174,A 0.000,B 0.000,C 90.000,E1 31.416} C_DIS
LIN {X -0.040,Y -219.139,Z 550.157,A 0.000,B 0.000,C 90.000,E1 28.359} C_DIS
LIN {X 0.049,Y -213.504,Z 550.140,A 0.000,B 0.000,C 90.000,E1 25.232} C_DIS
LIN {X 0.094,Y -208.716,Z 550.123,A 0.000,B 0.000,C 90.000,E1 22.078} C_DIS
LIN {X 0.023,Y -203.801,Z 550.101,A 0.000,B 0.000,C 90.000,E1 18.127} C_DIS
LIN {X 0.009,Y -199.978,Z 550.078,A 0.000,B 0.000,C 90.000,E1 14.120} C_DIS
LIN {X 0.006,Y -196.548,Z 550.047,A 0.000,B 0.000,C 90.000,E1 8.454} C_DIS
LIN {X 0.067,Y -195.461,Z 549.988,A 0.000,B 0.000,C 90.000,E1 357.879} C_DIS
LIN {X 0.029,Y -198.316,Z 549.952,A 0.000,B 0.000,C 90.000,E1 351.376} C_DIS
LIN {X 0.036,Y -201.992,Z 549.925,A 0.000,B 0.000,C 90.000,E1 346.520} C_DIS
LIN {X 0.030,Y -206.864,Z 549.898,A 0.000,B 0.000,C 90.000,E1 341.710} C_DIS
LIN {X 0.030,Y -211.806,Z 549.876,A 0.000,B 0.000,C 90.000,E1 337.741} C_DIS
LIN {X 0.014,Y -217.354,Z 549.855,A 0.000,B 0.000,C 90.000,E1 333.819} C_DIS
LIN {X -0.021,Y -223.457,Z 549.833,A 0.000,B 0.000,C 90.000,E1 329.950} C_DIS
LIN {X 0.113,Y -230.224,Z 549.812,A 0.000,B 0.000,C 90.000,E1 326.087} C_DIS
LIN {X 0.031,Y -236.035,Z 549.795,A 0.000,B 0.000,C 90.000,E1 323.084} C_DIS
LIN {X -0.075,Y -243.699,Z 549.774,A 0.000,B 0.000,C 90.000,E1 319.380} C_DIS
LIN {X 0.016,Y -252.334,Z 549.754,A 0.000,B 0.000,C 90.000,E1 315.688} C_DIS
LIN {X 0.027,Y -262.233,Z 549.734,A 0.000,B 0.000,C 90.000,E1 312.081} C_DIS
LIN {X 0.072,Y -273.504,Z 549.714,A 0.000,B 0.000,C 90.000,E1 308.543} C_DIS
LIN {X 0.016,Y -286.195,Z 549.695,A 0.000,B 0.000,C 90.000,E1 305.105} C_DIS
LIN {X -0.052,Y -300.262,Z 549.676,A 0.000,B 0.000,C 90.000,E1 301.750} C_DIS
LIN {X 0.175,Y -312.355,Z 549.662,A 0.000,B 0.000,C 90.000,E1 299.077} C_DIS
LIN {X -0.087,Y -326.941,Z 549.646,A 0.000,B 0.000,C 90.000,E1 296.232} C_DIS
LIN {X -0.053,Y -339.549,Z 549.633,A 0.000,B 0.000,C 90.000,E1 294.027} C_DIS
LIN {X 0.111,Y -351.456,Z 549.623,A 0.000,B 0.000,C 90.000,E1 292.153} C_DIS
LIN {X 0.133,Y -371.086,Z 549.608,A 0.000,B 0.000,C 90.000,E1 289.450} C_DIS
LIN {X -0.191,Y -387.516,Z 549.597,A 0.000,B 0.000,C 90.000,E1 287.457} C_DIS
LIN {X 0.098,Y -404.481,Z 549.586,A 0.000,B 0.000,C 90.000,E1 285.426} C_DIS
LIN {X 0.027,Y -419.121,Z 549.577,A 0.000,B 0.000,C 90.000,E1 283.772} C_DIS
LIN {X 0.040,Y -430.942,Z 549.569,A 0.000,B 0.000,C 90.000,E1 282.411} C_DIS
LIN {X -0.157,Y -439.964,Z 549.563,A 0.000,B 0.000,C 90.000,E1 281.366} C_DIS
LIN {X -0.163,Y -448.458,Z 549.557,A 0.000,B 0.000,C 90.000,E1 280.310} C_DIS
LIN {X -0.153,Y -456.316,Z 549.551,A 0.000,B 0.000,C 90.000,E1 279.265} C_DIS
LIN {X -0.049,Y -463.556,Z 549.546,A 0.000,B 0.000,C 90.000,E1 278.219} C_DIS
LIN {X -0.162,Y -468.502,Z 549.541,A 0.000,B 0.000,C 90.000,E1 277.466} C_DIS
LIN {X 0.173,Y -472.941,Z 549.537,A 0.000,B 0.000,C 90.000,E1 276.663} C_DIS
LIN {X 0.140,Y -476.865,Z 549.533,A 0.000,B 0.000,C 90.000,E1 275.910} C_DIS
LIN {X 0.087,Y -480.245,Z 549.529,A 0.000,B 0.000,C 90.000,E1 275.163} C_DIS
LIN {X 0.244,Y -482.113,Z 549.526,A 0.000,B 0.000,C 90.000,E1 274.645} C_DIS
LIN {X -0.112,Y -483.664,Z 549.523,A 0.000,B 0.000,C 90.000,E1 274.188} C_DIS
LIN {X 0.060,Y -484.912,Z 549.520,A 0.000,B 0.000,C 90.000,E1 273.669} C_DIS
LIN {X 0.212,Y -485.823,Z 549.518,A 0.000,B 0.000,C 90.000,E1 273.154} C_DIS
LIN {X -0.087,Y -486.419,Z 549.515,A 0.000,B 0.000,C 90.000,E1 272.694} C_DIS
LIN {X 0.080,Y -486.678,Z 549.512,A 0.000,B 0.000,C 90.000,E1 272.178} C_DIS
LIN {X -0.218,Y -486.563,Z 549.509,A 0.000,B 0.000,C 90.000,E1 271.718} C_DIS
LIN {X -0.045,Y -486.025,Z 549.507,A 0.000,B 0.000,C 90.000,E1 271.203} C_DIS
LIN {X 0.128,Y -485.038,Z 549.504,A 0.000,B 0.000,C 90.000,E1 270.688} C_DIS
LIN {X -0.185,Y -483.535,Z 549.501,A 0.000,B 0.000,C 90.000,E1 270.229} C_DIS
LIN {X -0.019,Y -481.396,Z 549.498,A 0.000,B 0.000,C 90.000,E1 269.714} C_DIS
LIN {X 0.136,Y -478.540,Z 549.496,A 0.000,B 0.000,C 90.000,E1 269.198} C_DIS
LIN {X -0.036,Y -476.824,Z 549.494,A 0.000,B 0.000,C 90.000,E1 268.969} C_DIS
LIN {X 0.087,Y -472.652,Z 549.491,A 0.000,B 0.000,C 90.000,E1 268.453} C_DIS
LIN {X -0.202,Y -467.337,Z 549.489,A 0.000,B 0.000,C 90.000,E1 267.993} C_DIS
LIN {X -0.182,Y -461.185,Z 549.486,A 0.000,B 0.000,C 90.000,E1 267.535} C_DIS
LIN {X -0.039,Y -457.701,Z 549.485,A 0.000,B 0.000,C 90.000,E1 267.306} C_DIS
LIN {X -0.084,Y -450.765,Z 549.483,A 0.000,B 0.000,C 90.000,E1 266.963} C_DIS
LIN {X -0.061,Y -443.698,Z 549.482,A 0.000,B 0.000,C 90.000,E1 266.674} C_DIS
LIN {X -0.140,Y -435.966,Z 549.480,A 0.000,B 0.000,C 90.000,E1 266.445} C_DIS
LIN {X -0.210,Y -427.707,Z 549.479,A 0.000,B 0.000,C 90.000,E1 266.274} C_DIS
LIN {X 0.110,Y -418.897,Z 549.478,A 0.000,B 0.000,C 90.000,E1 266.102} C_DIS
LIN {X 0.036,Y -409.115,Z 549.478,A 0.000,B 0.000,C 90.000,E1 266.045} C_DIS
LIN {X -0.019,Y -180.921,Z 549.478,A 0.000,B 0.000,C 90.000,E1 266.045} C_DIS
LIN {X 0.021,Y -180.865,Z 549.472,A 0.000,B 0.000,C 90.000,E1 265.008} C_DIS
LIN {X -0.076,Y -178.923,Z 549.443,A 0.000,B 0.000,C 90.000,E1 259.803} C_DIS
LIN {X -0.037,Y -175.969,Z 549.415,A 0.000,B 0.000,C 90.000,E1 254.700} C_DIS
LIN {X -0.043,Y -175.451,Z 549.410,A 0.000,B 0.000,C 90.000,E1 253.850} C_DIS
LIN {X -0.035,Y -172.205,Z 549.386,A 0.000,B 0.000,C 90.000,E1 249.571} C_DIS
LIN {X -0.057,Y -171.679,Z 549.382,A 0.000,B 0.000,C 90.000,E1 248.720} C_DIS
LIN {X -0.066,Y -167.905,Z 549.358,A 0.000,B 0.000,C 90.000,E1 244.409} C_DIS
LIN {X -0.047,Y -166.646,Z 549.348,A 0.000,B 0.000,C 90.000,E1 242.666} C_DIS
LIN {X 0.008,Y -162.630,Z 549.324,A 0.000,B 0.000,C 90.000,E1 238.280} C_DIS
LIN {X 0.067,Y -161.317,Z 549.314,A 0.000,B 0.000,C 90.000,E1 236.501} C_DIS
LIN {X -0.024,Y -157.314,Z 549.289,A 0.000,B 0.000,C 90.000,E1 232.110} C_DIS
LIN {X -0.090,Y -155.293,Z 549.275,A 0.000,B 0.000,C 90.000,E1 229.461} C_DIS
LIN {X 0.055,Y -151.654,Z 549.250,A 0.000,B 0.000,C 90.000,E1 224.919} C_DIS
LIN {X -0.007,Y -150.522,Z 549.240,A 0.000,B 0.000,C 90.000,E1 223.137} C_DIS
LIN {X 0.016,Y -147.246,Z 549.214,A 0.000,B 0.000,C 90.000,E1 218.588} C_DIS
LIN {X -0.019,Y -145.271,Z 549.194,A 0.000,B 0.000,C 90.000,E1 214.945} C_DIS
LIN {X 0.015,Y -142.378,Z 549.163,A 0.000,B 0.000,C 90.000,E1 209.411} C_DIS
LIN {X 0.064,Y -141.354,Z 549.148,A 0.000,B 0.000,C 90.000,E1 206.616} C_DIS
LIN {X 0.047,Y -139.341,Z 549.112,A 0.000,B 0.000,C 90.000,E1 200.120} C_DIS
LIN {X -0.034,Y -139.008,Z 549.102,A 0.000,B 0.000,C 90.000,E1 198.290} C_DIS
LIN {X 0.053,Y -138.340,Z 549.055,A 0.000,B 0.000,C 90.000,E1 189.849} C_DIS
LIN {X -0.063,Y -139.402,Z 549.008,A 0.000,B 0.000,C 90.000,E1 181.489} C_DIS
LIN {X -0.010,Y -141.308,Z 548.972,A 0.000,B 0.000,C 90.000,E1 174.951} C_DIS
LIN {X -0.052,Y -142.669,Z 548.956,A 0.000,B 0.000,C 90.000,E1 172.186} C_DIS
LIN {X 0.070,Y -145.018,Z 548.931,A 0.000,B 0.000,C 90.000,E1 167.521} C_DIS
LIN {X 0.027,Y -147.645,Z 548.910,A 0.000,B 0.000,C 90.000,E1 163.866} C_DIS
LIN {X -0.038,Y -150.279,Z 548.890,A 0.000,B 0.000,C 90.000,E1 160.242} C_DIS
LIN {X -0.024,Y -153.682,Z 548.870,A 0.000,B 0.000,C 90.000,E1 156.613} C_DIS
LIN {X 0.031,Y -157.096,Z 548.850,A 0.000,B 0.000,C 90.000,E1 152.999} C_DIS
LIN {X -0.031,Y -161.235,Z 548.830,A 0.000,B 0.000,C 90.000,E1 149.459} C_DIS
LIN {X 0.054,Y -163.322,Z 548.820,A 0.000,B 0.000,C 90.000,E1 147.661} C_DIS
LIN {X -0.075,Y -167.775,Z 548.801,A 0.000,B 0.000,C 90.000,E1 144.196} C_DIS
LIN {X 0.077,Y -171.589,Z 548.786,A 0.000,B 0.000,C 90.000,E1 141.537} C_DIS
LIN {X 0.008,Y -176.541,Z 548.767,A 0.000,B 0.000,C 90.000,E1 138.119} C_DIS
LIN {X 0.000,Y -180.839,Z 548.753,A 0.000,B 0.000,C 90.000,E1 135.567} C_DIS
LIN {X -0.015,Y -186.249,Z 548.734,A 0.000,B 0.000,C 90.000,E1 132.204} C_DIS
LIN {X 0.054,Y -191.350,Z 548.719,A 0.000,B 0.000,C 90.000,E1 129.402} C_DIS
LIN {X 0.031,Y -191.903,Z 548.717,A 0.000,B 0.000,C 90.000,E1 129.072} C_DIS
LIN {X 0.007,Y -289.122,Z 548.717,A 0.000,B 0.000,C 90.000,E1 129.072} C_DIS
LIN {X 0.001,Y -294.583,Z 548.716,A 0.000,B 0.000,C 90.000,E1 128.874} C_DIS
LIN {X -0.119,Y -297.407,Z 548.715,A 0.000,B 0.000,C 90.000,E1 128.669} C_DIS
LIN {X -0.045,Y -301.168,Z 548.712,A 0.000,B 0.000,C 90.000,E1 128.177} C_DIS
LIN {X 0.136,Y -302.987,Z 548.710,A 0.000,B 0.000,C 90.000,E1 127.810} C_DIS
LIN {X -0.107,Y -304.409,Z 548.708,A 0.000,B 0.000,C 90.000,E1 127.523} C_DIS
LIN {X -0.134,Y -306.437,Z 548.705,A 0.000,B 0.000,C 90.000,E1 126.870} C_DIS
LIN {X 0.048,Y -316.318,Z 548.687,A 0.000,B 0.000,C 90.000,E1 123.579} C_DIS
LIN {X -0.052,Y -326.519,Z 548.671,A 0.000,B 0.000,C 90.000,E1 120.718} C_DIS
LIN {X -0.090,Y -338.064,Z 548.655,A 0.000,B 0.000,C 90.000,E1 117.897} C_DIS
LIN {X 0.056,Y -351.052,Z 548.640,A 0.000,B 0.000,C 90.000,E1 115.103} C_DIS
LIN {X 0.042,Y -363.906,Z 548.626,A 0.000,B 0.000,C 90.000,E1 112.695} C_DIS
LIN {X -0.089,Y -378.089,Z 548.613,A 0.000,B 0.000,C 90.000,E1 110.355} C_DIS
LIN {X -0.131,Y -393.700,Z 548.600,A 0.000,B 0.000,C 90.000,E1 108.055} C_DIS
LIN {X -0.014,Y -410.859,Z 548.588,A 0.000,B 0.000,C 90.000,E1 105.788} C_DIS
LIN {X 0.031,Y -429.687,Z 548.576,A 0.000,B 0.000,C 90.000,E1 103.592} C_DIS
LIN {X -0.080,Y -449.731,Z 548.564,A 0.000,B 0.000,C 90.000,E1 101.535} C_DIS
LIN {X 0.103,Y -470.336,Z 548.553,A 0.000,B 0.000,C 90.000,E1 99.613} C_DIS
LIN {X 0.202,Y -475.551,Z 548.551,A 0.000,B 0.000,C 90.000,E1 99.151} C_DIS
LIN {X -0.162,Y -477.683,Z 548.550,A 0.000,B 0.000,C 90.000,E1 98.973} C_DIS
LIN {X 0.105,Y -479.490,Z 548.548,A 0.000,B 0.000,C 90.000,E1 98.690} C_DIS
LIN {X -0.029,Y -480.846,Z 548.547,A 0.000,B 0.000,C 90.000,E1 98.454} C_DIS
LIN {X 0.130,Y -482.546,Z 548.544,A 0.000,B 0.000,C 90.000,E1 97.936} C_DIS
LIN {X -0.117,Y -483.168,Z 548.541,A 0.000,B 0.000,C 90.000,E1 97.466} C_DIS
LIN {X 0.059,Y -482.815,Z 548.539,A 0.000,B 0.000,C 90.000,E1 96.947} C_DIS
LIN {X 0.239,Y -481.434,Z 548.536,A 0.000,B 0.000,C 90.000,E1 96.429} C_DIS
LIN {X 0.062,Y -480.287,Z 548.534,A 0.000,B 0.000,C 90.000,E1 96.201} C_DIS
LIN {X -0.063,Y -478.754,Z 548.533,A 0.000,B 0.000,C 90.000,E1 95.967} C_DIS
LIN {X 0.186,Y -461.432,Z 548.521,A 0.000,B 0.000,C 90.000,E1 93.669} C_DIS
LIN {X -0.212,Y -451.059,Z 548.512,A 0.000,B 0.000,C 90.000,E1 92.178} C_DIS
LIN {X -0.056,Y -435.791,Z 548.497,A 0.000,B 0.000,C 90.000,E1 89.542} C_DIS
LIN {X 0.001,Y -426.202,Z 548.489,A 0.000,B 0.000,C 90.000,E1 87.936} C_DIS
LIN {X 0.109,Y -413.497,Z 548.477,A 0.000,B 0.000,C 90.000,E1 85.755} C_DIS
LIN {X -0.057,Y -400.982,Z 548.464,A 0.000,B 0.000,C 90.000,E1 83.571} C_DIS
LIN {X -0.037,Y -388.722,Z 548.452,A 0.000,B 0.000,C 90.000,E1 81.319} C_DIS
LIN {X -0.188,Y -376.440,Z 548.439,A 0.000,B 0.000,C 90.000,E1 79.050} C_DIS
LIN {X -0.095,Y -359.997,Z 548.421,A 0.000,B 0.000,C 90.000,E1 75.811} C_DIS
LIN {X 0.118,Y -349.545,Z 548.408,A 0.000,B 0.000,C 90.000,E1 73.378} C_DIS
LIN {X -0.165,Y -339.087,Z 548.393,A 0.000,B 0.000,C 90.000,E1 70.678} C_DIS
LIN {X 0.017,Y -327.647,Z 548.374,A 0.000,B 0.000,C 90.000,E1 67.230} C_DIS
LIN {X -0.026,Y -317.992,Z 548.356,A 0.000,B 0.000,C 90.000,E1 64.076} C_DIS
LIN {X -0.053,Y -310.550,Z 548.342,A 0.000,B 0.000,C 90.000,E1 61.513} C_DIS
LIN {X 0.171,Y -303.112,Z 548.327,A 0.000,B 0.000,C 90.000,E1 58.869} C_DIS
LIN {X 0.030,Y -294.154,Z 548.309,A 0.000,B 0.000,C 90.000,E1 55.595} C_DIS
LIN {X -0.014,Y -287.327,Z 548.294,A 0.000,B 0.000,C 90.000,E1 52.924} C_DIS
LIN {X 0.027,Y -282.216,Z 548.283,A 0.000,B 0.000,C 90.000,E1 50.884} C_DIS
LIN {X -0.085,Y -278.556,Z 548.275,A 0.000,B 0.000,C 90.000,E1 49.542} C_DIS
LIN {X -0.058,Y -274.627,Z 548.268,A 0.000,B 0.000,C 90.000,E1 48.162} C_DIS
LIN {X -0.080,Y -270.402,Z 548.260,A 0.000,B 0.000,C 90.000,E1 46.782} C_DIS
LIN {X 0.026,Y -265.928,Z 548.252,A 0.000,B 0.000,C 90.000,E1 45.364} C_DIS
LIN {X -0.003,Y -257.643,Z 548.238,A 0.000,B 0.000,C 90.000,E1 42.894} C_DIS
LIN {X 0.030,Y -247.404,Z 548.220,A 0.000,B 0.000,C 90.000,E1 39.644} C_DIS
LIN {X 0.057,Y -236.846,Z 548.200,A 0.000,B 0.000,C 90.000,E1 35.964} C_DIS
LIN {X 0.102,Y -229.193,Z 548.183,A 0.000,B 0.000,C 90.000,E1 32.959} C_DIS
LIN {X 0.084,Y -222.304,Z 548.166,A 0.000,B 0.000,C 90.000,E1 29.922} C_DIS
LIN {X -0.046,Y -216.264,Z 548.149,A 0.000,B 0.000,C 90.000,E1 26.873} C_DIS
LIN {X -0.122,Y -211.039,Z 548.132,A 0.000,B 0.000,C 90.000,E1 23.770} C_DIS
LIN {X -0.091,Y -205.651,Z 548.110,A 0.000,B 0.000,C 90.000,E1 19.812} C_DIS
LIN {X 0.010,Y -201.375,Z 548.088,A 0.000,B 0.000,C 90.000,E1 15.788} C_DIS
LIN {X -0.002,Y -197.786,Z 548.061,A 0.000,B 0.000,C 90.000,E1 10.950} C_DIS
LIN {X 0.095,Y -195.229,Z 548.025,A 0.000,B 0.000,C 90.000,E1 4.416} C_DIS
LIN {X 0.080,Y -196.902,Z 547.966,A 0.000,B 0.000,C 90.000,E1 353.799} C_DIS
LIN {X -0.106,Y -200.564,Z 547.934,A 0.000,B 0.000,C 90.000,E1 348.173} C_DIS
LIN {X -0.027,Y -205.066,Z 547.907,A 0.000,B 0.000,C 90.000,E1 343.323} C_DIS
LIN {X -0.025,Y -209.710,Z 547.885,A 0.000,B 0.000,C 90.000,E1 339.337} C_DIS
LIN {X 0.109,Y -215.013,Z 547.863,A 0.000,B 0.000,C 90.000,E1 335.357} C_DIS
LIN {X -0.099,Y -220.909,Z 547.842,A 0.000,B 0.000,C 90.000,E1 331.513} C_DIS
LIN {X -0.091,Y -227.370,Z 547.820,A 0.000,B 0.000,C 90.000,E1 327.661} C_DIS
LIN {X -0.054,Y -233.051,Z 547.803,A 0.000,B 0.000,C 90.000,E1 324.609} C_DIS
LIN {X -0.117,Y -238.955,Z 547.787,A 0.000,B 0.000,C 90.000,E1 321.618} C_DIS
LIN {X 0.027,Y -246.993,Z 547.766,A 0.000,B 0.000,C 90.000,E1 317.877} C_DIS
LIN {X -0.151,Y -256.101,Z 547.746,A 0.000,B 0.000,C 90.000,E1 314.271} C_DIS
LIN {X 0.144,Y -265.476,Z 547.728,A 0.000,B 0.000,C 90.000,E1 310.987} C_DIS
LIN {X -0.053,Y -277.159,Z 547.708,A 0.000,B 0.000,C 90.000,E1 307.523} C_DIS
LIN {X 0.071,Y -290.226,Z 547.689,A 0.000,B 0.000,C 90.000,E1 304.072} C_DIS
LIN {X -0.020,Y -304.713,Z 547.671,A 0.000,B 0.000,C 90.000,E1 300.747} C_DIS
LIN {X -0.132,Y -320.238,Z 547.653,A 0.000,B 0.000,C 90.000,E1 297.513} C_DIS
LIN {X -0.112,Y -332.136,Z 547.640,A 0.000,B 0.000,C 90.000,E1 295.283} C_DIS
LIN {X 0.042,Y -343.354,Z 547.630,A 0.000,B 0.000,C 90.000,E1 293.387} C_DIS
LIN {X -0.145,Y -357.764,Z 547.618,A 0.000,B 0.000,C 90.000,E1 291.280} C_DIS
LIN {X 0.188,Y -373.414,Z 547.607,A 0.000,B 0.000,C 90.000,E1 289.141} C_DIS
LIN {X -0.055,Y -392.359,Z 547.594,A 0.000,B 0.000,C 90.000,E1 286.858} C_DIS
LIN {X -0.154,Y -409.392,Z 547.583,A 0.000,B 0.000,C 90.000,E1 284.898} C_DIS
LIN {X 0.130,Y -421.594,Z 547.575,A 0.000,B 0.000,C 90.000,E1 283.480} C_DIS
LIN {X 0.190,Y -433.328,Z 547.567,A 0.000,B 0.000,C 90.000,E1 282.119} C_DIS
LIN {X 0.026,Y -442.261,Z 547.562,A 0.000,B 0.000,C 90.000,E1 281.074} C_DIS
LIN {X 0.048,Y -450.586,Z 547.556,A 0.000,B 0.000,C 90.000,E1 280.018} C_DIS
LIN {X 0.086,Y -458.314,Z 547.550,A 0.000,B 0.000,C 90.000,E1 278.973} C_DIS
LIN {X -0.075,Y -463.699,Z 547.546,A 0.000,B 0.000,C 90.000,E1 278.219} C_DIS
LIN {X -0.186,Y -468.638,Z 547.541,A 0.000,B 0.000,C 90.000,E1 277.466} C_DIS
LIN {X 0.150,Y -473.072,Z 547.537,A 0.000,B 0.000,C 90.000,E1 276.663} C_DIS
LIN {X 0.118,Y -476.961,Z 547.533,A 0.000,B 0.000,C 90.000,E1 275.910} C_DIS
LIN {X 0.065,Y -480.330,Z 547.529,A 0.000,B 0.000,C 90.000,E1 275.163} C_DIS
LIN {X 0.223,Y -482.190,Z 547.526,A 0.000,B 0.000,C 90.000,E1 274.645} C_DIS
LIN {X -0.133,Y -483.721,Z 547.523,A 0.000,B 0.000,C 90.000,E1 274.188} C_DIS
LIN {X 0.040,Y -484.947,Z 547.520,A 0.000,B 0.000,C 90.000,E1 273.669} C_DIS
LIN {X 0.192,Y -485.826,Z 547.518,A 0.000,B 0.000,C 90.000,E1 273.154} C_DIS
LIN {X -0.107,Y -486.399,Z 547.515,A 0.000,B 0.000,C 90.000,E1 272.694} C_DIS
LIN {X 0.060,Y -486.638,Z 547.512,A 0.000,B 0.000,C 90.000,E1 272.178} C_DIS
LIN {X 0.248,Y -486.511,Z 547.509,A 0.000,B 0.000,C 90.000,E1 271.661} C_DIS
LIN {X -0.065,Y -485.973,Z 547.507,A 0.000,B 0.000,C 90.000,E1 271.203} C_DIS
LIN {X 0.107,Y -484.994,Z 547.504,A 0.000,B 0.000,C 90.000,E1 270.688} C_DIS
LIN {X -0.205,Y -483.489,Z 547.501,A 0.000,B 0.000,C 90.000,E1 270.229} C_DIS
LIN {X -0.040,Y -481.346,Z 547.498,A 0.000,B 0.000,C 90.000,E1 269.714} C_DIS
LIN {X 0.115,Y -478.510,Z 547.496,A 0.000,B 0.000,C 90.000,E1 269.198} C_DIS
LIN {X -0.228,Y -474.804,Z 547.493,A 0.000,B 0.000,C 90.000,E1 268.740} C_DIS
LIN {X -0.113,Y -470.050,Z 547.490,A 0.000,B 0.000,C 90.000,E1 268.224} C_DIS
LIN {X 0.222,Y -467.253,Z 547.489,A 0.000,B 0.000,C 90.000,E1 267.936} C_DIS
LIN {X 0.074,Y -464.127,Z 547.487,A 0.000,B 0.000,C 90.000,E1 267.707} C_DIS
LIN {X 0.205,Y -461.045,Z 547.486,A 0.000,B 0.000,C 90.000,E1 267.478} C_DIS
LIN {X -0.127,Y -454.222,Z 547.484,A 0.000,B 0.000,C 90.000,E1 267.135} C_DIS
LIN {X 0.114,Y -447.148,Z 547.482,A 0.000,B 0.000,C 90.000,E1 266.788} C_DIS
LIN {X -0.166,Y -439.816,Z 547.481,A 0.000,B 0.000,C 90.000,E1 266.560} C_DIS
LIN {X 0.217,Y -435.669,Z 547.480,A 0.000,B 0.000,C 90.000,E1 266.388} C_DIS
LIN {X 0.129,Y -427.225,Z 547.479,A 0.000,B 0.000,C 90.000,E1 266.216} C_DIS
LIN {X 0.004,Y -417.595,Z 547.478,A 0.000,B 0.000,C 90.000,E1 266.102} C_DIS
LIN {X -0.051,Y -405.420,Z 547.478,A 0.000,B 0.000,C 90.000,E1 266.045} C_DIS
LIN {X -0.057,Y -180.921,Z 547.478,A 0.000,B 0.000,C 90.000,E1 266.045} C_DIS
LIN {X -0.015,Y -180.862,Z 547.472,A 0.000,B 0.000,C 90.000,E1 265.008} C_DIS
LIN {X 0.064,Y -178.918,Z 547.443,A 0.000,B 0.000,C 90.000,E1 259.746} C_DIS
LIN {X -0.026,Y -175.964,Z 547.415,A 0.000,B 0.000,C 90.000,E1 254.685} C_DIS
LIN {X 0.089,Y -175.442,Z 547.410,A 0.000,B 0.000,C 90.000,E1 253.795} C_DIS
